LIN {X 0,Y 574.072,Z 399.932,A -85,B 0,C 180,E1 -2018.319,E2 -2018.319} C_VEL
LIN {X 0,Y 573.881,Z 501.404,A -85,B 0,C 180,E1 -2019.612,E2 -2019.612} C_VEL
LIN {X 0,Y 573.788,Z 514.414,A -85,B 0,C 180,E1 -2019.919,E2 -2019.919} C_VEL
LIN {X 0,Y 573.675,Z 527.236,A -85,B 0,C 180,E1 -2020.373,E2 -2020.373} C_VEL
LIN {X 0,Y 573.572,Z 539.532,A -85,B 0,C 180,E1 -2020.968,E2 -2020.968} C_VEL
LIN {X 0,Y 573.479,Z 550.065,A -85,B 0,C 180,E1 -2021.62,E2 -2021.62} C_VEL
LIN {X 0,Y 573.322,Z 560.171,A -85,B 0,C 180,E1 -2022.393,E2 -2022.393} C_VEL
LIN {X 0,Y 573.221,Z 570.379,A -85,B 0,C 180,E1 -2023.361,E2 -2023.361} C_VEL
LIN {X 0,Y 573.135,Z 578.736,A -85,B 0,C 180,E1 -2024.344,E2 -2024.344} C_VEL
LIN {X 0,Y 573.071,Z 585.667,A -85,B 0,C 180,E1 -2025.341,E2 -2025.341} C_VEL
LIN {X 0,Y 573.025,Z 591.385,A -85,B 0,C 180,E1 -2026.355,E2 -2026.355} C_VEL
LIN {X 0,Y 573.008,Z 596.786,A -85,B 0,C 180,E1 -2027.578,E2 -2027.578} C_VEL
LIN {X 0,Y 572.995,Z 599.936,A -85,B 0,C 180,E1 -2028.521,E2 -2028.521} C_VEL
LIN {X 0,Y 572.949,Z 602.391,A -85,B 0,C 180,E1 -2029.51,E2 -2029.51} C_VEL
LIN {X 0,Y 572.921,Z 604.15,A -85,B 0,C 180,E1 -2030.608,E2 -2030.608} C_VEL
LIN {X 0,Y 572.93,Z 604.936,A -85,B 0,C 180,E1 -2031.728,E2 -2031.728} C_VEL
LIN {X 0,Y 572.956,Z 604.58,A -85,B 0,C 180,E1 -2033.055,E2 -2033.055} C_VEL
LIN {X 0,Y 572.93,Z 603.35,A -85,B 0,C 180,E1 -2034.058,E2 -2034.058} C_VEL
LIN {X 0,Y 572.989,Z 600.789,A -85,B 0,C 180,E1 -2035.265,E2 -2035.265} C_VEL
LIN {X 0,Y 572.998,Z 596.77,A -85,B 0,C 180,E1 -2036.517,E2 -2036.517} C_VEL
LIN {X 0,Y 573.082,Z 591.054,A -85,B 0,C 180,E1 -2037.799,E2 -2037.799} C_VEL
LIN {X 0,Y 573.123,Z 584.06,A -85,B 0,C 180,E1 -2039,E2 -2039} C_VEL
LIN {X 0,Y 573.181,Z 576.654,A -85,B 0,C 180,E1 -2040.01,E2 -2040.01} C_VEL
LIN {X 0,Y 573.27,Z 567.371,A -85,B 0,C 180,E1 -2041.036,E2 -2041.036} C_VEL
LIN {X 0,Y 573.355,Z 557.054,A -85,B 0,C 180,E1 -2041.953,E2 -2041.953} C_VEL
LIN {X 0,Y 573.484,Z 545.995,A -85,B 0,C 180,E1 -2042.739,E2 -2042.739} C_VEL
LIN {X 0,Y 573.617,Z 535.091,A -85,B 0,C 180,E1 -2043.356,E2 -2043.356} C_VEL
LIN {X 0,Y 573.709,Z 523.101,A -85,B 0,C 180,E1 -2043.88,E2 -2043.88} C_VEL
LIN {X 0,Y 573.83,Z 510.167,A -85,B 0,C 180,E1 -2044.288,E2 -2044.288} C_VEL
LIN {X 0,Y 573.889,Z 497.236,A -85,B 0,C 180,E1 -2044.546,E2 -2044.546} C_VEL
LIN {X 0,Y 574.062,Z 398.701,A -85,B 0,C 180,E1 -2045.786,E2 -2045.786} C_VEL
LIN {X 0,Y 573.309,Z 394.131,A -85,B 0,C 180,E1 -2045.873,E2 -2045.873} C_VEL
LIN {X 0,Y 573.457,Z 376.545,A -85,B 0,C 180,E1 -2048.923,E2 -2048.923} C_VEL
LIN {X 0,Y 573.564,Z 362.34,A -85,B 0,C 180,E1 -2051.422,E2 -2051.422} C_VEL
LIN {X 0,Y 573.289,Z 360.075,A -85,B 0,C 180,E1 -2051.875,E2 -2051.875} C_VEL
LIN {X 0,Y 573.241,Z 360.081,A -85,B 0,C 180,E1 -2054.351,E2 -2054.351} C_VEL
LIN {X 0,Y 573.241,Z 360.084,A -85,B 0,C 180,E1 -2056.529,E2 -2056.529} C_VEL
LIN {X 0,Y 573.269,Z 360.077,A -85,B 0,C 180,E1 -2058.744,E2 -2058.744} C_VEL
LIN {X 0,Y 573.288,Z 360.068,A -85,B 0,C 180,E1 -2061.54,E2 -2061.54} C_VEL
LIN {X 0,Y 573.294,Z 360.076,A -85,B 0,C 180,E1 -2064.371,E2 -2064.371} C_VEL
LIN {X 0,Y 573.316,Z 360.067,A -85,B 0,C 180,E1 -2067.892,E2 -2067.892} C_VEL
LIN {X 0,Y 573.336,Z 360.066,A -85,B 0,C 180,E1 -2070.701,E2 -2070.701} C_VEL
LIN {X 0,Y 573.309,Z 360.068,A -85,B 0,C 180,E1 -2072.81,E2 -2072.81} C_VEL
LIN {X 0,Y 573.292,Z 360.069,A -85,B 0,C 180,E1 -2075.627,E2 -2075.627} C_VEL
LIN {X 0,Y 573.285,Z 360.074,A -85,B 0,C 180,E1 -2078.458,E2 -2078.458} C_VEL
LIN {X 0,Y 573.275,Z 360.07,A -85,B 0,C 180,E1 -2081.311,E2 -2081.311} C_VEL
LIN {X 0,Y 573.284,Z 360.073,A -85,B 0,C 180,E1 -2084.423,E2 -2084.423} C_VEL
LIN {X 0,Y 573.261,Z 360.071,A -85,B 0,C 180,E1 -2087.11,E2 -2087.11} C_VEL
LIN {X 0,Y 573.242,Z 360.082,A -85,B 0,C 180,E1 -2090.076,E2 -2090.076} C_VEL
LIN {X 0,Y 573.235,Z 360.078,A -85,B 0,C 180,E1 -2092.337,E2 -2092.337} C_VEL
LIN {X 0,Y 573.255,Z 360.075,A -85,B 0,C 180,E1 -2095.409,E2 -2095.409} C_VEL
LIN {X 0,Y 573.252,Z 360.079,A -85,B 0,C 180,E1 -2098.028,E2 -2098.028} C_VEL
LIN {X 0,Y 573.241,Z 360.074,A -85,B 0,C 180,E1 -2100.884,E2 -2100.884} C_VEL
LIN {X 0,Y 573.259,Z 360.079,A -85,B 0,C 180,E1 -2103.523,E2 -2103.523} C_VEL
LIN {X 0,Y 573.259,Z 360.075,A -85,B 0,C 180,E1 -2106.047,E2 -2106.047} C_VEL
LIN {X 0,Y 573.246,Z 360.073,A -85,B 0,C 180,E1 -2108.7,E2 -2108.7} C_VEL
LIN {X 0,Y 573.25,Z 360.082,A -85,B 0,C 180,E1 -2111.595,E2 -2111.595} C_VEL
LIN {X 0,Y 573.234,Z 360.076,A -85,B 0,C 180,E1 -2114.332,E2 -2114.332} C_VEL
LIN {X 0,Y 573.245,Z 360.083,A -85,B 0,C 180,E1 -2117.356,E2 -2117.356} C_VEL
LIN {X 0,Y 573.287,Z 360.256,A -85,B 0,C 180,E1 -2118.288,E2 -2118.288} C_VEL
LIN {X 0,Y 573.535,Z 365.736,A -85,B 0,C 180,E1 -2119.269,E2 -2119.269} C_VEL
LIN {X 0,Y 573.423,Z 380.934,A -85,B 0,C 180,E1 -2121.932,E2 -2121.932} C_VEL
LIN {X 0,Y 573.275,Z 394.135,A -85,B 0,C 180,E1 -2124.217,E2 -2124.217} C_VEL
LIN {X 0,Y 574.068,Z 400.409,A -85,B 0,C 180,E1 -2124.325,E2 -2124.325} C_VEL
LIN {X 0,Y 573.887,Z 500.332,A -85,B 0,C 180,E1 -2125.597,E2 -2125.597} C_VEL
LIN {X 0,Y 573.82,Z 512.126,A -85,B 0,C 180,E1 -2125.857,E2 -2125.857} C_VEL
LIN {X 0,Y 573.706,Z 525.236,A -85,B 0,C 180,E1 -2126.292,E2 -2126.292} C_VEL
LIN {X 0,Y 573.58,Z 537.36,A -85,B 0,C 180,E1 -2126.853,E2 -2126.853} C_VEL
LIN {X 0,Y 573.467,Z 548.11,A -85,B 0,C 180,E1 -2127.492,E2 -2127.492} C_VEL
LIN {X 0,Y 573.346,Z 558.978,A -85,B 0,C 180,E1 -2128.294,E2 -2128.294} C_VEL
LIN {X 0,Y 573.265,Z 569.447,A -85,B 0,C 180,E1 -2129.265,E2 -2129.265} C_VEL
LIN {X 0,Y 573.129,Z 577.631,A -85,B 0,C 180,E1 -2130.207,E2 -2130.207} C_VEL
LIN {X 0,Y 573.111,Z 584.91,A -85,B 0,C 180,E1 -2131.228,E2 -2131.228} C_VEL
LIN {X 0,Y 573.022,Z 591.708,A -85,B 0,C 180,E1 -2132.419,E2 -2132.419} C_VEL
LIN {X 0,Y 573.03,Z 596.673,A -85,B 0,C 180,E1 -2133.546,E2 -2133.546} C_VEL
LIN {X 0,Y 572.989,Z 600.113,A -85,B 0,C 180,E1 -2134.577,E2 -2134.577} C_VEL
LIN {X 0,Y 572.959,Z 602.073,A -85,B 0,C 180,E1 -2135.351,E2 -2135.351} C_VEL
LIN {X 0,Y 572.924,Z 603.479,A -85,B 0,C 180,E1 -2136.121,E2 -2136.121} C_VEL
LIN {X 0,Y 572.967,Z 604.451,A -85,B 0,C 180,E1 -2136.915,E2 -2136.915} C_VEL
LIN {X 0,Y 572.938,Z 604.921,A -85,B 0,C 180,E1 -2137.65,E2 -2137.65} C_VEL
LIN {X 0,Y 572.97,Z 604.761,A -85,B 0,C 180,E1 -2138.778,E2 -2138.778} C_VEL
LIN {X 0,Y 572.969,Z 603.567,A -85,B 0,C 180,E1 -2139.913,E2 -2139.913} C_VEL
LIN {X 0,Y 572.956,Z 601.885,A -85,B 0,C 180,E1 -2140.817,E2 -2140.817} C_VEL
LIN {X 0,Y 572.991,Z 599.33,A -85,B 0,C 180,E1 -2141.774,E2 -2141.774} C_VEL
LIN {X 0,Y 572.994,Z 595.309,A -85,B 0,C 180,E1 -2142.88,E2 -2142.88} C_VEL
LIN {X 0,Y 573.044,Z 590.075,A -85,B 0,C 180,E1 -2143.981,E2 -2143.981} C_VEL
LIN {X 0,Y 573.091,Z 583.522,A -85,B 0,C 180,E1 -2145.076,E2 -2145.076} C_VEL
LIN {X 0,Y 573.174,Z 575.367,A -85,B 0,C 180,E1 -2146.166,E2 -2146.166} C_VEL
LIN {X 0,Y 573.277,Z 567.009,A -85,B 0,C 180,E1 -2147.071,E2 -2147.071} C_VEL
LIN {X 0,Y 573.342,Z 557.888,A -85,B 0,C 180,E1 -2147.882,E2 -2147.882} C_VEL
LIN {X 0,Y 573.449,Z 548.891,A -85,B 0,C 180,E1 -2148.546,E2 -2148.546} C_VEL
LIN {X 0,Y 573.551,Z 538.875,A -85,B 0,C 180,E1 -2149.154,E2 -2149.154} C_VEL
LIN {X 0,Y 573.661,Z 528.069,A -85,B 0,C 180,E1 -2149.678,E2 -2149.678} C_VEL
LIN {X 0,Y 573.77,Z 515.206,A -85,B 0,C 180,E1 -2150.148,E2 -2150.148} C_VEL
LIN {X 0,Y 573.895,Z 502.194,A -85,B 0,C 180,E1 -2150.462,E2 -2150.462} C_VEL
LIN {X 0,Y 573.934,Z 468.796,A -85,B 0,C 180,E1 -2150.907,E2 -2150.907} C_VEL
LIN {X 0,Y 574.041,Z 398.761,A -85,B 0,C 180,E1 -2151.786,E2 -2151.786} C_VEL
LIN {X 0,Y 573.334,Z 394.179,A -85,B 0,C 180,E1 -2151.864,E2 -2151.864} C_VEL
LIN {X 0,Y 573.428,Z 376.67,A -85,B 0,C 180,E1 -2154.902,E2 -2154.902} C_VEL
LIN {X 0,Y 573.566,Z 363.645,A -85,B 0,C 180,E1 -2157.191,E2 -2157.191} C_VEL
LIN {X 0,Y 573.275,Z 360.076,A -85,B 0,C 180,E1 -2157.848,E2 -2157.848} C_VEL
LIN {X 0,Y 573.312,Z 360.069,A -85,B 0,C 180,E1 -2160,E2 -2160} C_VEL
LIN {X 0,Y 573.306,Z 360.073,A -85,B 0,C 180,E1 -2162.811,E2 -2162.811} C_VEL
LIN {X 0,Y 573.285,Z 360.07,A -85,B 0,C 180,E1 -2165.628,E2 -2165.628} C_VEL
LIN {X 0,Y 573.298,Z 360.076,A -85,B 0,C 180,E1 -2168.459,E2 -2168.459} C_VEL
LIN {X 0,Y 573.289,Z 360.069,A -85,B 0,C 180,E1 -2171.312,E2 -2171.312} C_VEL
LIN {X 0,Y 573.271,Z 360.077,A -85,B 0,C 180,E1 -2174.425,E2 -2174.425} C_VEL
LIN {X 0,Y 573.252,Z 360.073,A -85,B 0,C 180,E1 -2177.112,E2 -2177.112} C_VEL
LIN {X 0,Y 573.25,Z 360.082,A -85,B 0,C 180,E1 -2180.077,E2 -2180.077} C_VEL
LIN {X 0,Y 573.262,Z 360.072,A -85,B 0,C 180,E1 -2183.154,E2 -2183.154} C_VEL
LIN {X 0,Y 573.284,Z 360.073,A -85,B 0,C 180,E1 -2186.189,E2 -2186.189} C_VEL
LIN {X 0,Y 573.235,Z 360.076,A -85,B 0,C 180,E1 -2188.565,E2 -2188.565} C_VEL
LIN {X 0,Y 573.234,Z 360.077,A -85,B 0,C 180,E1 -2190.993,E2 -2190.993} C_VEL
LIN {X 0,Y 573.28,Z 360.079,A -85,B 0,C 180,E1 -2193.529,E2 -2193.529} C_VEL
LIN {X 0,Y 573.253,Z 360.075,A -85,B 0,C 180,E1 -2196.049,E2 -2196.049} C_VEL
LIN {X 0,Y 573.242,Z 360.075,A -85,B 0,C 180,E1 -2198.702,E2 -2198.702} C_VEL
LIN {X 0,Y 573.247,Z 360.079,A -85,B 0,C 180,E1 -2201.597,E2 -2201.597} C_VEL
LIN {X 0,Y 573.233,Z 360.075,A -85,B 0,C 180,E1 -2204.334,E2 -2204.334} C_VEL
LIN {X 0,Y 573.234,Z 360.082,A -85,B 0,C 180,E1 -2207.359,E2 -2207.359} C_VEL
LIN {X 0,Y 573.244,Z 360.075,A -85,B 0,C 180,E1 -2210.394,E2 -2210.394} C_VEL
LIN {X 0,Y 573.253,Z 360.081,A -85,B 0,C 180,E1 -2213.079,E2 -2213.079} C_VEL
LIN {X 0,Y 573.272,Z 360.071,A -85,B 0,C 180,E1 -2215.673,E2 -2215.673} C_VEL
LIN {X 0,Y 573.247,Z 360.075,A -85,B 0,C 180,E1 -2218.186,E2 -2218.186} C_VEL
LIN {X 0,Y 573.268,Z 360.079,A -85,B 0,C 180,E1 -2220.636,E2 -2220.636} C_VEL
LIN {X 0,Y 573.269,Z 360.072,A -85,B 0,C 180,E1 -2223.502,E2 -2223.502} C_VEL
LIN {X 0,Y 573.232,Z 360.081,A -85,B 0,C 180,E1 -2226.136,E2 -2226.136} C_VEL
LIN {X 0,Y 573.254,Z 360.175,A -85,B 0,C 180,E1 -2226.937,E2 -2226.937} C_VEL
LIN {X 0,Y 574.015,Z 365.028,A -85,B 0,C 180,E1 -2227.695,E2 -2227.695} C_VEL
LIN {X 0,Y 573.747,Z 385.178,A -85,B 0,C 180,E1 -2230.688,E2 -2230.688} C_VEL
LIN {X 0,Y 573.562,Z 404.099,A -85,B 0,C 180,E1 -2233.454,E2 -2233.454} C_VEL
LIN {X 0,Y 573.381,Z 422.8,A -85,B 0,C 180,E1 -2236.15,E2 -2236.15} C_VEL
LIN {X 0,Y 574.12,Z 428.592,A -85,B 0,C 180,E1 -2236.259,E2 -2236.259} C_VEL
LIN {X 0,Y 573.908,Z 530.999,A -85,B 0,C 180,E1 -2237.559,E2 -2237.559} C_VEL
LIN {X 0,Y 573.777,Z 544.254,A -85,B 0,C 180,E1 -2237.87,E2 -2237.87} C_VEL
LIN {X 0,Y 573.703,Z 556.4,A -85,B 0,C 180,E1 -2238.295,E2 -2238.295} C_VEL
LIN {X 0,Y 573.593,Z 568.646,A -85,B 0,C 180,E1 -2238.874,E2 -2238.874} C_VEL
LIN {X 0,Y 573.434,Z 580.216,A -85,B 0,C 180,E1 -2239.586,E2 -2239.586} C_VEL
LIN {X 0,Y 573.327,Z 590.612,A -85,B 0,C 180,E1 -2240.386,E2 -2240.386} C_VEL
LIN {X 0,Y 573.24,Z 599.123,A -85,B 0,C 180,E1 -2241.186,E2 -2241.186} C_VEL
LIN {X 0,Y 573.16,Z 606.969,A -85,B 0,C 180,E1 -2242.072,E2 -2242.072} C_VEL
LIN {X 0,Y 573.073,Z 614.586,A -85,B 0,C 180,E1 -2243.127,E2 -2243.127} C_VEL
LIN {X 0,Y 573.07,Z 621.685,A -85,B 0,C 180,E1 -2244.371,E2 -2244.371} C_VEL
LIN {X 0,Y 573.028,Z 626.376,A -85,B 0,C 180,E1 -2245.428,E2 -2245.428} C_VEL
LIN {X 0,Y 573.022,Z 629.96,A -85,B 0,C 180,E1 -2246.485,E2 -2246.485} C_VEL
LIN {X 0,Y 572.959,Z 631.81,A -85,B 0,C 180,E1 -2247.189,E2 -2247.189} C_VEL
LIN {X 0,Y 572.938,Z 633.2,A -85,B 0,C 180,E1 -2247.892,E2 -2247.892} C_VEL
LIN {X 0,Y 572.941,Z 634.786,A -85,B 0,C 180,E1 -2249.298,E2 -2249.298} C_VEL
LIN {X 0,Y 572.938,Z 635,A -85,B 0,C 180,E1 -2250.001,E2 -2250.001} C_VEL
LIN {X 0,Y 572.946,Z 634.185,A -85,B 0,C 180,E1 -2251.407,E2 -2251.407} C_VEL
LIN {X 0,Y 572.938,Z 633.198,A -85,B 0,C 180,E1 -2252.11,E2 -2252.11} C_VEL
LIN {X 0,Y 572.959,Z 631.808,A -85,B 0,C 180,E1 -2252.813,E2 -2252.813} C_VEL
LIN {X 0,Y 573.014,Z 628.893,A -85,B 0,C 180,E1 -2253.869,E2 -2253.869} C_VEL
LIN {X 0,Y 572.963,Z 624.945,A -85,B 0,C 180,E1 -2254.926,E2 -2254.926} C_VEL
LIN {X 0,Y 573.064,Z 618.872,A -85,B 0,C 180,E1 -2256.161,E2 -2256.161} C_VEL
LIN {X 0,Y 573.12,Z 612.232,A -85,B 0,C 180,E1 -2257.222,E2 -2257.222} C_VEL
LIN {X 0,Y 573.199,Z 603.983,A -85,B 0,C 180,E1 -2258.284,E2 -2258.284} C_VEL
LIN {X 0,Y 573.287,Z 595.529,A -85,B 0,C 180,E1 -2259.171,E2 -2259.171} C_VEL
LIN {X 0,Y 573.421,Z 585.087,A -85,B 0,C 180,E1 -2260.059,E2 -2260.059} C_VEL
LIN {X 0,Y 573.528,Z 573.342,A -85,B 0,C 180,E1 -2260.859,E2 -2260.859} C_VEL
LIN {X 0,Y 573.655,Z 562.264,A -85,B 0,C 180,E1 -2261.448,E2 -2261.448} C_VEL
LIN {X 0,Y 573.759,Z 549.148,A -85,B 0,C 180,E1 -2261.975,E2 -2261.975} C_VEL
LIN {X 0,Y 573.866,Z 536.485,A -85,B 0,C 180,E1 -2262.331,E2 -2262.331} C_VEL
LIN {X 0,Y 573.928,Z 523.244,A -85,B 0,C 180,E1 -2262.555,E2 -2262.555} C_VEL
LIN {X 0,Y 573.944,Z 426.655,A -85,B 0,C 180,E1 -2263.77,E2 -2263.77} C_VEL
LIN {X 0,Y 573.379,Z 422.787,A -85,B 0,C 180,E1 -2263.852,E2 -2263.852} C_VEL
LIN {X 0,Y 573.547,Z 402.884,A -85,B 0,C 180,E1 -2266.724,E2 -2266.724} C_VEL
LIN {X 0,Y 573.735,Z 384.58,A -85,B 0,C 180,E1 -2269.401,E2 -2269.401} C_VEL
LIN {X 0,Y 574.002,Z 365.015,A -85,B 0,C 180,E1 -2272.307,E2 -2272.307} C_VEL
LIN {X 0,Y 573.24,Z 360.085,A -85,B 0,C 180,E1 -2273.1,E2 -2273.1} C_VEL
LIN {X 0,Y 573.261,Z 360.081,A -85,B 0,C 180,E1 -2275.411,E2 -2275.411} C_VEL
LIN {X 0,Y 573.256,Z 360.075,A -85,B 0,C 180,E1 -2278.029,E2 -2278.029} C_VEL
LIN {X 0,Y 573.244,Z 360.079,A -85,B 0,C 180,E1 -2280.884,E2 -2280.884} C_VEL
LIN {X 0,Y 573.268,Z 360.076,A -85,B 0,C 180,E1 -2283.524,E2 -2283.524} C_VEL
LIN {X 0,Y 573.221,Z 360.077,A -85,B 0,C 180,E1 -2286.052,E2 -2286.052} C_VEL
LIN {X 0,Y 573.255,Z 360.077,A -85,B 0,C 180,E1 -2288.701,E2 -2288.701} C_VEL
LIN {X 0,Y 573.234,Z 360.078,A -85,B 0,C 180,E1 -2291.593,E2 -2291.593} C_VEL
LIN {X 0,Y 573.241,Z 360.076,A -85,B 0,C 180,E1 -2294.334,E2 -2294.334} C_VEL
LIN {X 0,Y 573.246,Z 360.077,A -85,B 0,C 180,E1 -2297.359,E2 -2297.359} C_VEL
LIN {X 0,Y 573.243,Z 360.076,A -85,B 0,C 180,E1 -2300.392,E2 -2300.392} C_VEL
LIN {X 0,Y 573.257,Z 360.078,A -85,B 0,C 180,E1 -2303.078,E2 -2303.078} C_VEL
LIN {X 0,Y 573.271,Z 360.07,A -85,B 0,C 180,E1 -2305.671,E2 -2305.671} C_VEL
LIN {X 0,Y 573.245,Z 360.076,A -85,B 0,C 180,E1 -2308.185,E2 -2308.185} C_VEL
LIN {X 0,Y 573.268,Z 360.079,A -85,B 0,C 180,E1 -2310.634,E2 -2310.634} C_VEL
LIN {X 0,Y 573.24,Z 360.073,A -85,B 0,C 180,E1 -2313.508,E2 -2313.508} C_VEL
LIN {X 0,Y 573.235,Z 360.078,A -85,B 0,C 180,E1 -2316.135,E2 -2316.135} C_VEL
LIN {X 0,Y 573.255,Z 360.074,A -85,B 0,C 180,E1 -2319.174,E2 -2319.174} C_VEL
LIN {X 0,Y 573.222,Z 360.075,A -85,B 0,C 180,E1 -2321.411,E2 -2321.411} C_VEL
LIN {X 0,Y 573.254,Z 360.073,A -85,B 0,C 180,E1 -2323.622,E2 -2323.622} C_VEL
LIN {X 0,Y 573.277,Z 360.07,A -85,B 0,C 180,E1 -2325.807,E2 -2325.807} C_VEL
LIN {X 0,Y 573.269,Z 360.073,A -85,B 0,C 180,E1 -2328.745,E2 -2328.745} C_VEL
LIN {X 0,Y 573.288,Z 360.069,A -85,B 0,C 180,E1 -2331.541,E2 -2331.541} C_VEL
LIN {X 0,Y 573.295,Z 360.074,A -85,B 0,C 180,E1 -2334.372,E2 -2334.372} C_VEL
LIN {X 0,Y 573.316,Z 360.07,A -85,B 0,C 180,E1 -2337.892,E2 -2337.892} C_VEL
LIN {X 0,Y 573.335,Z 360.063,A -85,B 0,C 180,E1 -2340.702,E2 -2340.702} C_VEL
LIN {X 0,Y 573.311,Z 360.066,A -85,B 0,C 180,E1 -2342.811,E2 -2342.811} C_VEL
LIN {X 0,Y 573.296,Z 360.072,A -85,B 0,C 180,E1 -2345.628,E2 -2345.628} C_VEL
LIN {X 0,Y 573.289,Z 360.07,A -85,B 0,C 180,E1 -2348.46,E2 -2348.46} C_VEL
LIN {X 0,Y 573.278,Z 360.072,A -85,B 0,C 180,E1 -2351.312,E2 -2351.312} C_VEL
LIN {X 0,Y 573.287,Z 360.07,A -85,B 0,C 180,E1 -2354.424,E2 -2354.424} C_VEL
LIN {X 0,Y 573.264,Z 360.073,A -85,B 0,C 180,E1 -2357.112,E2 -2357.112} C_VEL
LIN {X 0,Y 573.257,Z 360.076,A -85,B 0,C 180,E1 -2360.077,E2 -2360.077} C_VEL
LIN {X 0,Y 573.241,Z 360.077,A -85,B 0,C 180,E1 -2363.099,E2 -2363.099} C_VEL
LIN {X 0,Y 573.255,Z 360.073,A -85,B 0,C 180,E1 -2364.387,E2 -2364.387} C_VEL
LIN {X 0,Y 572.63,Z 360.154,A -85,B 0,C 180,E1 -2364.974,E2 -2364.974} C_VEL
LIN {X 0,Y 569.791,Z 360.512,A -85,B 0,C 180,E1 -2365.925,E2 -2365.925} C_VEL
LIN {X 0,Y 567.357,Z 360.818,A -85,B 0,C 180,E1 -2366.691,E2 -2366.691} C_VEL
LIN {X 0,Y 566.296,Z 360.948,A -85,B 0,C 180,E1 -2367.282,E2 -2367.282} C_VEL
LIN {X 0,Y 566.203,Z 360.957,A -85,B 0,C 180,E1 -2367.482,E2 -2367.482} C_VEL
LIN {X 0,Y 566.207,Z 360.958,A -85,B 0,C 180,E1 -2369.769,E2 -2369.769} C_VEL
LIN {X 0,Y 566.23,Z 361.071,A -85,B 0,C 180,E1 -2372.178,E2 -2372.178} C_VEL
LIN {X 0,Y 566.543,Z 366.033,A -85,B 0,C 180,E1 -2373.081,E2 -2373.081} C_VEL
LIN {X 0,Y 566.377,Z 382.226,A -85,B 0,C 180,E1 -2375.954,E2 -2375.954} C_VEL
LIN {X 0,Y 566.257,Z 394.162,A -85,B 0,C 180,E1 -2378.047,E2 -2378.047} C_VEL
LIN {X 0,Y 567.172,Z 400.604,A -85,B 0,C 180,E1 -2378.158,E2 -2378.158} C_VEL
LIN {X 0,Y 566.943,Z 501.598,A -85,B 0,C 180,E1 -2379.461,E2 -2379.461} C_VEL
LIN {X 0,Y 566.835,Z 514.735,A -85,B 0,C 180,E1 -2379.778,E2 -2379.778} C_VEL
LIN {X 0,Y 566.716,Z 526.907,A -85,B 0,C 180,E1 -2380.214,E2 -2380.214} C_VEL
LIN {X 0,Y 566.595,Z 539.544,A -85,B 0,C 180,E1 -2380.83,E2 -2380.83} C_VEL
LIN {X 0,Y 566.465,Z 551.449,A -85,B 0,C 180,E1 -2381.588,E2 -2381.588} C_VEL
LIN {X 0,Y 566.258,Z 562.13,A -85,B 0,C 180,E1 -2382.444,E2 -2382.444} C_VEL
LIN {X 0,Y 566.182,Z 570.576,A -85,B 0,C 180,E1 -2383.273,E2 -2383.273} C_VEL
LIN {X 0,Y 566.078,Z 578.913,A -85,B 0,C 180,E1 -2384.27,E2 -2384.27} C_VEL
LIN {X 0,Y 566.011,Z 585.787,A -85,B 0,C 180,E1 -2385.276,E2 -2385.276} C_VEL
LIN {X 0,Y 565.945,Z 592.441,A -85,B 0,C 180,E1 -2386.498,E2 -2386.498} C_VEL
LIN {X 0,Y 565.914,Z 596.69,A -85,B 0,C 180,E1 -2387.497,E2 -2387.497} C_VEL
LIN {X 0,Y 565.923,Z 599.027,A -85,B 0,C 180,E1 -2388.17,E2 -2388.17} C_VEL
LIN {X 0,Y 565.846,Z 601.944,A -85,B 0,C 180,E1 -2389.257,E2 -2389.257} C_VEL
LIN {X 0,Y 565.852,Z 603.889,A -85,B 0,C 180,E1 -2390.359,E2 -2390.359} C_VEL
LIN {X 0,Y 565.835,Z 604.911,A -85,B 0,C 180,E1 -2391.608,E2 -2391.608} C_VEL
LIN {X 0,Y 565.816,Z 604.853,A -85,B 0,C 180,E1 -2392.65,E2 -2392.65} C_VEL
LIN {X 0,Y 565.826,Z 603.728,A -85,B 0,C 180,E1 -2393.838,E2 -2393.838} C_VEL
LIN {X 0,Y 565.879,Z 601.155,A -85,B 0,C 180,E1 -2395.158,E2 -2395.158} C_VEL
LIN {X 0,Y 565.925,Z 597.713,A -85,B 0,C 180,E1 -2396.31,E2 -2396.31} C_VEL
LIN {X 0,Y 565.951,Z 592.347,A -85,B 0,C 180,E1 -2397.611,E2 -2397.611} C_VEL
LIN {X 0,Y 566.001,Z 585.959,A -85,B 0,C 180,E1 -2398.785,E2 -2398.785} C_VEL
LIN {X 0,Y 566.104,Z 578.954,A -85,B 0,C 180,E1 -2399.814,E2 -2399.814} C_VEL
LIN {X 0,Y 566.197,Z 570.325,A -85,B 0,C 180,E1 -2400.843,E2 -2400.843} C_VEL
LIN {X 0,Y 566.309,Z 560.612,A -85,B 0,C 180,E1 -2401.779,E2 -2401.779} C_VEL
LIN {X 0,Y 566.444,Z 550.474,A -85,B 0,C 180,E1 -2402.572,E2 -2402.572} C_VEL
LIN {X 0,Y 566.614,Z 539.526,A -85,B 0,C 180,E1 -2403.26,E2 -2403.26} C_VEL
LIN {X 0,Y 566.724,Z 527.948,A -85,B 0,C 180,E1 -2403.831,E2 -2403.831} C_VEL
LIN {X 0,Y 566.842,Z 515.148,A -85,B 0,C 180,E1 -2404.3,E2 -2404.3} C_VEL
LIN {X 0,Y 566.944,Z 502.434,A -85,B 0,C 180,E1 -2404.613,E2 -2404.613} C_VEL
LIN {X 0,Y 567.034,Z 471.171,A -85,B 0,C 180,E1 -2405.036,E2 -2405.036} C_VEL
LIN {X 0,Y 567.071,Z 399.012,A -85,B 0,C 180,E1 -2405.955,E2 -2405.955} C_VEL
LIN {X 0,Y 566.29,Z 394.166,A -85,B 0,C 180,E1 -2406.042,E2 -2406.042} C_VEL
LIN {X 0,Y 566.425,Z 376.763,A -85,B 0,C 180,E1 -2409.1,E2 -2409.1} C_VEL
LIN {X 0,Y 566.576,Z 364.003,A -85,B 0,C 180,E1 -2411.372,E2 -2411.372} C_VEL
LIN {X 0,Y 566.26,Z 360.951,A -85,B 0,C 180,E1 -2411.97,E2 -2411.97} C_VEL
LIN {X 0,Y 566.205,Z 360.957,A -85,B 0,C 180,E1 -2414.89,E2 -2414.89} C_VEL
LIN {X 0,Y 566.249,Z 360.946,A -85,B 0,C 180,E1 -2417.818,E2 -2417.818} C_VEL
LIN {X 0,Y 566.212,Z 360.956,A -85,B 0,C 180,E1 -2420.713,E2 -2420.713} C_VEL
LIN {X 0,Y 566.23,Z 360.948,A -85,B 0,C 180,E1 -2423.197,E2 -2423.197} C_VEL
LIN {X 0,Y 566.189,Z 360.953,A -85,B 0,C 180,E1 -2425.728,E2 -2425.728} C_VEL
LIN {X 0,Y 566.287,Z 360.943,A -85,B 0,C 180,E1 -2427.865,E2 -2427.865} C_VEL
LIN {X 0,Y 566.307,Z 360.942,A -85,B 0,C 180,E1 -2430.71,E2 -2430.71} C_VEL
LIN {X 0,Y 566.275,Z 360.944,A -85,B 0,C 180,E1 -2432.845,E2 -2432.845} C_VEL
LIN {X 0,Y 566.261,Z 360.946,A -85,B 0,C 180,E1 -2435.697,E2 -2435.697} C_VEL
LIN {X 0,Y 566.229,Z 360.951,A -85,B 0,C 180,E1 -2438.565,E2 -2438.565} C_VEL
LIN {X 0,Y 566.245,Z 360.947,A -85,B 0,C 180,E1 -2441.453,E2 -2441.453} C_VEL
LIN {X 0,Y 566.237,Z 360.95,A -85,B 0,C 180,E1 -2444.506,E2 -2444.506} C_VEL
LIN {X 0,Y 566.204,Z 360.952,A -85,B 0,C 180,E1 -2447.33,E2 -2447.33} C_VEL
LIN {X 0,Y 566.208,Z 360.954,A -85,B 0,C 180,E1 -2450.336,E2 -2450.336} C_VEL
LIN {X 0,Y 566.173,Z 360.956,A -85,B 0,C 180,E1 -2453.281,E2 -2453.281} C_VEL
LIN {X 0,Y 566.214,Z 360.958,A -85,B 0,C 180,E1 -2455.748,E2 -2455.748} C_VEL
LIN {X 0,Y 566.201,Z 360.954,A -85,B 0,C 180,E1 -2458.201,E2 -2458.201} C_VEL
LIN {X 0,Y 566.192,Z 360.952,A -85,B 0,C 180,E1 -2460.591,E2 -2460.591} C_VEL
LIN {X 0,Y 566.226,Z 360.949,A -85,B 0,C 180,E1 -2463.1,E2 -2463.1} C_VEL
LIN {X 0,Y 566.211,Z 360.959,A -85,B 0,C 180,E1 -2465.687,E2 -2465.687} C_VEL
LIN {X 0,Y 566.212,Z 360.949,A -85,B 0,C 180,E1 -2468.558,E2 -2468.558} C_VEL
LIN {X 0,Y 566.208,Z 360.954,A -85,B 0,C 180,E1 -2471.135,E2 -2471.135} C_VEL
LIN {X 0,Y 566.195,Z 360.955,A -85,B 0,C 180,E1 -2474.034,E2 -2474.034} C_VEL
LIN {X 0,Y 566.204,Z 360.956,A -85,B 0,C 180,E1 -2477.081,E2 -2477.081} C_VEL
LIN {X 0,Y 566.277,Z 361.149,A -85,B 0,C 180,E1 -2478.194,E2 -2478.194} C_VEL
LIN {X 0,Y 566.541,Z 366.546,A -85,B 0,C 180,E1 -2479.173,E2 -2479.173} C_VEL
LIN {X 0,Y 566.374,Z 383.071,A -85,B 0,C 180,E1 -2482.103,E2 -2482.103} C_VEL
LIN {X 0,Y 566.263,Z 394.133,A -85,B 0,C 180,E1 -2484.042,E2 -2484.042} C_VEL
LIN {X 0,Y 567.178,Z 399.933,A -85,B 0,C 180,E1 -2484.149,E2 -2484.149} C_VEL
LIN {X 0,Y 566.957,Z 500.764,A -85,B 0,C 180,E1 -2485.45,E2 -2485.45} C_VEL
LIN {X 0,Y 566.857,Z 513.412,A -85,B 0,C 180,E1 -2485.739,E2 -2485.739} C_VEL
LIN {X 0,Y 566.749,Z 526.141,A -85,B 0,C 180,E1 -2486.182,E2 -2486.182} C_VEL
LIN {X 0,Y 566.609,Z 537.294,A -85,B 0,C 180,E1 -2486.711,E2 -2486.711} C_VEL
LIN {X 0,Y 566.469,Z 548.004,A -85,B 0,C 180,E1 -2487.354,E2 -2487.354} C_VEL
LIN {X 0,Y 566.325,Z 557.62,A -85,B 0,C 180,E1 -2488.064,E2 -2488.064} C_VEL
LIN {X 0,Y 566.22,Z 567.122,A -85,B 0,C 180,E1 -2488.916,E2 -2488.916} C_VEL
LIN {X 0,Y 566.096,Z 576.945,A -85,B 0,C 180,E1 -2490.02,E2 -2490.02} C_VEL
LIN {X 0,Y 566.037,Z 584.23,A -85,B 0,C 180,E1 -2491.038,E2 -2491.038} C_VEL
LIN {X 0,Y 565.942,Z 590.121,A -85,B 0,C 180,E1 -2492.044,E2 -2492.044} C_VEL
LIN {X 0,Y 565.928,Z 594.856,A -85,B 0,C 180,E1 -2493.046,E2 -2493.046} C_VEL
LIN {X 0,Y 565.918,Z 599.224,A -85,B 0,C 180,E1 -2494.236,E2 -2494.236} C_VEL
LIN {X 0,Y 565.861,Z 601.399,A -85,B 0,C 180,E1 -2495.045,E2 -2495.045} C_VEL
LIN {X 0,Y 565.827,Z 602.987,A -85,B 0,C 180,E1 -2495.802,E2 -2495.802} C_VEL
LIN {X 0,Y 565.845,Z 604.354,A -85,B 0,C 180,E1 -2496.792,E2 -2496.792} C_VEL
LIN {X 0,Y 565.83,Z 604.952,A -85,B 0,C 180,E1 -2498.122,E2 -2498.122} C_VEL
LIN {X 0,Y 565.884,Z 604.688,A -85,B 0,C 180,E1 -2498.889,E2 -2498.889} C_VEL
LIN {X 0,Y 565.855,Z 603.994,A -85,B 0,C 180,E1 -2499.649,E2 -2499.649} C_VEL
LIN {X 0,Y 565.863,Z 602.194,A -85,B 0,C 180,E1 -2500.716,E2 -2500.716} C_VEL
LIN {X 0,Y 565.908,Z 599.027,A -85,B 0,C 180,E1 -2501.912,E2 -2501.912} C_VEL
LIN {X 0,Y 565.922,Z 595.122,A -85,B 0,C 180,E1 -2502.982,E2 -2502.982} C_VEL
LIN {X 0,Y 565.95,Z 589.593,A -85,B 0,C 180,E1 -2504.145,E2 -2504.145} C_VEL
LIN {X 0,Y 566.043,Z 582.7,A -85,B 0,C 180,E1 -2505.291,E2 -2505.291} C_VEL
LIN {X 0,Y 566.118,Z 574.637,A -85,B 0,C 180,E1 -2506.357,E2 -2506.357} C_VEL
LIN {X 0,Y 566.239,Z 566.073,A -85,B 0,C 180,E1 -2507.273,E2 -2507.273} C_VEL
LIN {X 0,Y 566.342,Z 556.77,A -85,B 0,C 180,E1 -2508.094,E2 -2508.094} C_VEL
LIN {X 0,Y 566.445,Z 548.159,A -85,B 0,C 180,E1 -2508.726,E2 -2508.726} C_VEL
LIN {X 0,Y 566.643,Z 537.477,A -85,B 0,C 180,E1 -2509.368,E2 -2509.368} C_VEL
LIN {X 0,Y 566.774,Z 524.897,A -85,B 0,C 180,E1 -2509.958,E2 -2509.958} C_VEL
LIN {X 0,Y 566.842,Z 512.035,A -85,B 0,C 180,E1 -2510.387,E2 -2510.387} C_VEL
LIN {X 0,Y 566.96,Z 500.947,A -85,B 0,C 180,E1 -2510.636,E2 -2510.636} C_VEL
LIN {X 0,Y 567.087,Z 399.252,A -85,B 0,C 180,E1 -2511.952,E2 -2511.952} C_VEL
LIN {X 0,Y 566.276,Z 394.042,A -85,B 0,C 180,E1 -2512.064,E2 -2512.064} C_VEL
LIN {X 0,Y 566.403,Z 377.236,A -85,B 0,C 180,E1 -2515.017,E2 -2515.017} C_VEL
LIN {X 0,Y 566.571,Z 365.207,A -85,B 0,C 180,E1 -2517.156,E2 -2517.156} C_VEL
LIN {X 0,Y 566.266,Z 360.949,A -85,B 0,C 180,E1 -2517.955,E2 -2517.955} C_VEL
LIN {X 0,Y 566.3,Z 360.948,A -85,B 0,C 180,E1 -2520.711,E2 -2520.711} C_VEL
LIN {X 0,Y 566.271,Z 360.949,A -85,B 0,C 180,E1 -2522.846,E2 -2522.846} C_VEL
LIN {X 0,Y 566.253,Z 360.947,A -85,B 0,C 180,E1 -2525.698,E2 -2525.698} C_VEL
LIN {X 0,Y 566.239,Z 360.953,A -85,B 0,C 180,E1 -2528.566,E2 -2528.566} C_VEL
LIN {X 0,Y 566.241,Z 360.947,A -85,B 0,C 180,E1 -2531.454,E2 -2531.454} C_VEL
LIN {X 0,Y 566.224,Z 360.953,A -85,B 0,C 180,E1 -2534.507,E2 -2534.507} C_VEL
LIN {X 0,Y 566.197,Z 360.953,A -85,B 0,C 180,E1 -2537.332,E2 -2537.332} C_VEL
LIN {X 0,Y 566.212,Z 360.954,A -85,B 0,C 180,E1 -2540.337,E2 -2540.337} C_VEL
LIN {X 0,Y 566.225,Z 360.951,A -85,B 0,C 180,E1 -2543.402,E2 -2543.402} C_VEL
LIN {X 0,Y 566.22,Z 360.958,A -85,B 0,C 180,E1 -2545.749,E2 -2545.749} C_VEL
LIN {X 0,Y 566.199,Z 360.955,A -85,B 0,C 180,E1 -2548.204,E2 -2548.204} C_VEL
LIN {X 0,Y 566.187,Z 360.953,A -85,B 0,C 180,E1 -2550.593,E2 -2550.593} C_VEL
LIN {X 0,Y 566.221,Z 360.952,A -85,B 0,C 180,E1 -2553.102,E2 -2553.102} C_VEL
LIN {X 0,Y 566.204,Z 360.958,A -85,B 0,C 180,E1 -2555.689,E2 -2555.689} C_VEL
LIN {X 0,Y 566.208,Z 360.951,A -85,B 0,C 180,E1 -2558.56,E2 -2558.56} C_VEL
LIN {X 0,Y 566.205,Z 360.957,A -85,B 0,C 180,E1 -2561.137,E2 -2561.137} C_VEL
LIN {X 0,Y 566.194,Z 360.953,A -85,B 0,C 180,E1 -2564.036,E2 -2564.036} C_VEL
LIN {X 0,Y 566.195,Z 360.96,A -85,B 0,C 180,E1 -2567.084,E2 -2567.084} C_VEL
LIN {X 0,Y 566.222,Z 360.95,A -85,B 0,C 180,E1 -2569.804,E2 -2569.804} C_VEL
LIN {X 0,Y 566.195,Z 360.956,A -85,B 0,C 180,E1 -2572.6,E2 -2572.6} C_VEL
LIN {X 0,Y 566.219,Z 360.955,A -85,B 0,C 180,E1 -2575.184,E2 -2575.184} C_VEL
LIN {X 0,Y 566.231,Z 360.948,A -85,B 0,C 180,E1 -2577.745,E2 -2577.745} C_VEL
LIN {X 0,Y 566.226,Z 360.952,A -85,B 0,C 180,E1 -2580.324,E2 -2580.324} C_VEL
LIN {X 0,Y 566.233,Z 360.95,A -85,B 0,C 180,E1 -2583.336,E2 -2583.336} C_VEL
LIN {X 0,Y 566.198,Z 360.955,A -85,B 0,C 180,E1 -2585.821,E2 -2585.821} C_VEL
LIN {X 0,Y 566.208,Z 361.122,A -85,B 0,C 180,E1 -2586.798,E2 -2586.798} C_VEL
LIN {X 0,Y 567.07,Z 366.19,A -85,B 0,C 180,E1 -2587.599,E2 -2587.599} C_VEL
LIN {X 0,Y 566.788,Z 386.047,A -85,B 0,C 180,E1 -2590.571,E2 -2590.571} C_VEL
LIN {X 0,Y 566.58,Z 404.253,A -85,B 0,C 180,E1 -2593.266,E2 -2593.266} C_VEL
LIN {X 0,Y 566.386,Z 422.8,A -85,B 0,C 180,E1 -2595.976,E2 -2595.976} C_VEL
LIN {X 0,Y 567.214,Z 429.374,A -85,B 0,C 180,E1 -2596.098,E2 -2596.098} C_VEL
LIN {X 0,Y 566.988,Z 530.999,A -85,B 0,C 180,E1 -2597.405,E2 -2597.405} C_VEL
LIN {X 0,Y 566.855,Z 543.492,A -85,B 0,C 180,E1 -2597.697,E2 -2597.697} C_VEL
LIN {X 0,Y 566.744,Z 556.402,A -85,B 0,C 180,E1 -2598.149,E2 -2598.149} C_VEL
LIN {X 0,Y 566.594,Z 567.454,A -85,B 0,C 180,E1 -2598.671,E2 -2598.671} C_VEL
LIN {X 0,Y 566.491,Z 578.923,A -85,B 0,C 180,E1 -2599.367,E2 -2599.367} C_VEL
LIN {X 0,Y 566.332,Z 589.552,A -85,B 0,C 180,E1 -2600.176,E2 -2600.176} C_VEL
LIN {X 0,Y 566.206,Z 599.123,A -85,B 0,C 180,E1 -2601.075,E2 -2601.075} C_VEL
LIN {X 0,Y 566.111,Z 606.969,A -85,B 0,C 180,E1 -2601.973,E2 -2601.973} C_VEL
LIN {X 0,Y 566,Z 614.628,A -85,B 0,C 180,E1 -2603.048,E2 -2603.048} C_VEL
LIN {X 0,Y 566.003,Z 621.685,A -85,B 0,C 180,E1 -2604.3,E2 -2604.3} C_VEL
LIN {X 0,Y 565.933,Z 626.376,A -85,B 0,C 180,E1 -2605.371,E2 -2605.371} C_VEL
LIN {X 0,Y 565.927,Z 629.96,A -85,B 0,C 180,E1 -2606.441,E2 -2606.441} C_VEL
LIN {X 0,Y 565.878,Z 631.81,A -85,B 0,C 180,E1 -2607.153,E2 -2607.153} C_VEL
LIN {X 0,Y 565.846,Z 634.186,A -85,B 0,C 180,E1 -2608.578,E2 -2608.578} C_VEL
LIN {X 0,Y 565.839,Z 635,A -85,B 0,C 180,E1 -2610.001,E2 -2610.001} C_VEL
LIN {X 0,Y 565.846,Z 634.185,A -85,B 0,C 180,E1 -2611.424,E2 -2611.424} C_VEL
LIN {X 0,Y 565.878,Z 631.808,A -85,B 0,C 180,E1 -2612.848,E2 -2612.848} C_VEL
LIN {X 0,Y 565.926,Z 628.893,A -85,B 0,C 180,E1 -2613.917,E2 -2613.917} C_VEL
LIN {X 0,Y 565.878,Z 624.945,A -85,B 0,C 180,E1 -2614.988,E2 -2614.988} C_VEL
LIN {X 0,Y 566.002,Z 619.862,A -85,B 0,C 180,E1 -2616.059,E2 -2616.059} C_VEL
LIN {X 0,Y 566.041,Z 613.462,A -85,B 0,C 180,E1 -2617.133,E2 -2617.133} C_VEL
LIN {X 0,Y 566.133,Z 605.471,A -85,B 0,C 180,E1 -2618.209,E2 -2618.209} C_VEL
LIN {X 0,Y 566.229,Z 597.327,A -85,B 0,C 180,E1 -2619.106,E2 -2619.106} C_VEL
LIN {X 0,Y 566.343,Z 587.39,A -85,B 0,C 180,E1 -2620.006,E2 -2620.006} C_VEL
LIN {X 0,Y 566.53,Z 576.278,A -85,B 0,C 180,E1 -2620.808,E2 -2620.808} C_VEL
LIN {X 0,Y 566.614,Z 565.159,A -85,B 0,C 180,E1 -2621.448,E2 -2621.448} C_VEL
LIN {X 0,Y 566.771,Z 552.961,A -85,B 0,C 180,E1 -2621.988,E2 -2621.988} C_VEL
LIN {X 0,Y 566.909,Z 540.142,A -85,B 0,C 180,E1 -2622.394,E2 -2622.394} C_VEL
LIN {X 0,Y 566.988,Z 528.05,A -85,B 0,C 180,E1 -2622.643,E2 -2622.643} C_VEL
LIN {X 0,Y 567.038,Z 427.298,A -85,B 0,C 180,E1 -2623.933,E2 -2623.933} C_VEL
LIN {X 0,Y 566.378,Z 422.787,A -85,B 0,C 180,E1 -2624.026,E2 -2624.026} C_VEL
LIN {X 0,Y 566.592,Z 401.707,A -85,B 0,C 180,E1 -2627.109,E2 -2627.109} C_VEL
LIN {X 0,Y 566.852,Z 381.387,A -85,B 0,C 180,E1 -2630.125,E2 -2630.125} C_VEL
LIN {X 0,Y 567.053,Z 366.132,A -85,B 0,C 180,E1 -2632.403,E2 -2632.403} C_VEL
LIN {X 0,Y 566.215,Z 360.961,A -85,B 0,C 180,E1 -2633.235,E2 -2633.235} C_VEL
LIN {X 0,Y 566.22,Z 360.954,A -85,B 0,C 180,E1 -2635.749,E2 -2635.749} C_VEL
LIN {X 0,Y 566.208,Z 360.952,A -85,B 0,C 180,E1 -2638.203,E2 -2638.203} C_VEL
LIN {X 0,Y 566.205,Z 360.958,A -85,B 0,C 180,E1 -2641.078,E2 -2641.078} C_VEL
LIN {X 0,Y 566.218,Z 360.952,A -85,B 0,C 180,E1 -2643.735,E2 -2643.735} C_VEL
LIN {X 0,Y 566.206,Z 360.953,A -85,B 0,C 180,E1 -2646.57,E2 -2646.57} C_VEL
LIN {X 0,Y 566.228,Z 360.951,A -85,B 0,C 180,E1 -2649.687,E2 -2649.687} C_VEL
LIN {X 0,Y 566.207,Z 360.959,A -85,B 0,C 180,E1 -2652.918,E2 -2652.918} C_VEL
LIN {X 0,Y 566.204,Z 360.951,A -85,B 0,C 180,E1 -2656.049,E2 -2656.049} C_VEL
LIN {X 0,Y 566.209,Z 360.954,A -85,B 0,C 180,E1 -2659.215,E2 -2659.215} C_VEL
LIN {X 0,Y 566.188,Z 360.953,A -85,B 0,C 180,E1 -2661.637,E2 -2661.637} C_VEL
LIN {X 0,Y 566.167,Z 360.958,A -85,B 0,C 180,E1 -2664.308,E2 -2664.308} C_VEL
LIN {X 0,Y 566.225,Z 360.956,A -85,B 0,C 180,E1 -2666.898,E2 -2666.898} C_VEL
LIN {X 0,Y 566.185,Z 360.953,A -85,B 0,C 180,E1 -2669.407,E2 -2669.407} C_VEL
LIN {X 0,Y 566.2,Z 360.952,A -85,B 0,C 180,E1 -2671.857,E2 -2671.857} C_VEL
LIN {X 0,Y 566.215,Z 360.953,A -85,B 0,C 180,E1 -2674.251,E2 -2674.251} C_VEL
LIN {X 0,Y 566.177,Z 360.96,A -85,B 0,C 180,E1 -2676.719,E2 -2676.719} C_VEL
LIN {X 0,Y 566.218,Z 360.95,A -85,B 0,C 180,E1 -2679.663,E2 -2679.663} C_VEL
LIN {X 0,Y 566.204,Z 360.957,A -85,B 0,C 180,E1 -2682.668,E2 -2682.668} C_VEL
LIN {X 0,Y 566.239,Z 360.946,A -85,B 0,C 180,E1 -2685.627,E2 -2685.627} C_VEL
LIN {X 0,Y 566.24,Z 360.949,A -85,B 0,C 180,E1 -2688.675,E2 -2688.675} C_VEL
LIN {X 0,Y 566.232,Z 360.948,A -85,B 0,C 180,E1 -2691.434,E2 -2691.434} C_VEL
LIN {X 0,Y 566.264,Z 360.952,A -85,B 0,C 180,E1 -2694.302,E2 -2694.302} C_VEL
LIN {X 0,Y 566.287,Z 360.945,A -85,B 0,C 180,E1 -2697.866,E2 -2697.866} C_VEL
LIN {X 0,Y 566.306,Z 360.939,A -85,B 0,C 180,E1 -2700.711,E2 -2700.711} C_VEL
LIN {X 0,Y 566.277,Z 360.942,A -85,B 0,C 180,E1 -2702.846,E2 -2702.846} C_VEL
LIN {X 0,Y 566.264,Z 360.949,A -85,B 0,C 180,E1 -2705.698,E2 -2705.698} C_VEL
LIN {X 0,Y 566.233,Z 360.948,A -85,B 0,C 180,E1 -2708.566,E2 -2708.566} C_VEL
LIN {X 0,Y 566.248,Z 360.95,A -85,B 0,C 180,E1 -2711.454,E2 -2711.454} C_VEL
LIN {X 0,Y 566.24,Z 360.947,A -85,B 0,C 180,E1 -2714.507,E2 -2714.507} C_VEL
LIN {X 0,Y 566.205,Z 360.955,A -85,B 0,C 180,E1 -2717.332,E2 -2717.332} C_VEL
LIN {X 0,Y 566.218,Z 360.951,A -85,B 0,C 180,E1 -2720.337,E2 -2720.337} C_VEL
LIN {X 0,Y 566.178,Z 360.96,A -85,B 0,C 180,E1 -2723.282,E2 -2723.282} C_VEL
LIN {X 0,Y 566.22,Z 360.956,A -85,B 0,C 180,E1 -2725.749,E2 -2725.749} C_VEL
LIN {X 0,Y 566.203,Z 360.957,A -85,B 0,C 180,E1 -2727.482,E2 -2727.482} C_VEL
LIN {X 0,Y 565.517,Z 361.04,A -85,B 0,C 180,E1 -2728.076,E2 -2728.076} C_VEL
LIN {X 0,Y 562.653,Z 361.398,A -85,B 0,C 180,E1 -2729.039,E2 -2729.039} C_VEL
LIN {X 0,Y 560.249,Z 361.699,A -85,B 0,C 180,E1 -2729.815,E2 -2729.815} C_VEL
LIN {X 0,Y 559.225,Z 361.823,A -85,B 0,C 180,E1 -2730.414,E2 -2730.414} C_VEL
LIN {X 0,Y 559.145,Z 361.833,A -85,B 0,C 180,E1 -2730.617,E2 -2730.617} C_VEL
LIN {X 0,Y 559.192,Z 361.923,A -85,B 0,C 180,E1 -2732.047,E2 -2732.047} C_VEL
LIN {X 0,Y 559.57,Z 366.475,A -85,B 0,C 180,E1 -2732.902,E2 -2732.902} C_VEL
LIN {X 0,Y 559.35,Z 383.49,A -85,B 0,C 180,E1 -2735.973,E2 -2735.973} C_VEL
LIN {X 0,Y 559.222,Z 394.161,A -85,B 0,C 180,E1 -2737.867,E2 -2737.867} C_VEL
LIN {X 0,Y 560.303,Z 401.509,A -85,B 0,C 180,E1 -2737.996,E2 -2737.996} C_VEL
LIN {X 0,Y 560.025,Z 501.163,A -85,B 0,C 180,E1 -2739.295,E2 -2739.295} C_VEL
LIN {X 0,Y 559.91,Z 514.164,A -85,B 0,C 180,E1 -2739.606,E2 -2739.606} C_VEL
LIN {X 0,Y 559.774,Z 527.064,A -85,B 0,C 180,E1 -2740.072,E2 -2740.072} C_VEL
LIN {X 0,Y 559.603,Z 539.225,A -85,B 0,C 180,E1 -2740.671,E2 -2740.671} C_VEL
LIN {X 0,Y 559.45,Z 550.495,A -85,B 0,C 180,E1 -2741.386,E2 -2741.386} C_VEL
LIN {X 0,Y 559.271,Z 561.314,A -85,B 0,C 180,E1 -2742.25,E2 -2742.25} C_VEL
LIN {X 0,Y 559.139,Z 570.874,A -85,B 0,C 180,E1 -2743.195,E2 -2743.195} C_VEL
LIN {X 0,Y 559.027,Z 579.31,A -85,B 0,C 180,E1 -2744.225,E2 -2744.225} C_VEL
LIN {X 0,Y 558.926,Z 586.071,A -85,B 0,C 180,E1 -2745.238,E2 -2745.238} C_VEL
LIN {X 0,Y 558.873,Z 591.522,A -85,B 0,C 180,E1 -2746.239,E2 -2746.239} C_VEL
LIN {X 0,Y 558.84,Z 595.867,A -85,B 0,C 180,E1 -2747.225,E2 -2747.225} C_VEL
LIN {X 0,Y 558.815,Z 600.487,A -85,B 0,C 180,E1 -2748.624,E2 -2748.624} C_VEL
LIN {X 0,Y 558.768,Z 601.785,A -85,B 0,C 180,E1 -2749.152,E2 -2749.152} C_VEL
LIN {X 0,Y 558.77,Z 603.543,A -85,B 0,C 180,E1 -2750.107,E2 -2750.107} C_VEL
LIN {X 0,Y 558.733,Z 604.735,A -85,B 0,C 180,E1 -2751.249,E2 -2751.249} C_VEL
LIN {X 0,Y 558.726,Z 604.926,A -85,B 0,C 180,E1 -2752.416,E2 -2752.416} C_VEL
LIN {X 0,Y 558.729,Z 603.881,A -85,B 0,C 180,E1 -2753.758,E2 -2753.758} C_VEL
LIN {X 0,Y 558.772,Z 602.001,A -85,B 0,C 180,E1 -2754.84,E2 -2754.84} C_VEL
LIN {X 0,Y 558.82,Z 598.587,A -85,B 0,C 180,E1 -2756.104,E2 -2756.104} C_VEL
LIN {X 0,Y 558.86,Z 593.577,A -85,B 0,C 180,E1 -2757.413,E2 -2757.413} C_VEL
LIN {X 0,Y 558.917,Z 588.279,A -85,B 0,C 180,E1 -2758.472,E2 -2758.472} C_VEL
LIN {X 0,Y 558.997,Z 581.233,A -85,B 0,C 180,E1 -2759.599,E2 -2759.599} C_VEL
LIN {X 0,Y 559.114,Z 573.08,A -85,B 0,C 180,E1 -2760.644,E2 -2760.644} C_VEL
LIN {X 0,Y 559.234,Z 563.869,A -85,B 0,C 180,E1 -2761.607,E2 -2761.607} C_VEL
LIN {X 0,Y 559.431,Z 553.211,A -85,B 0,C 180,E1 -2762.504,E2 -2762.504} C_VEL
LIN {X 0,Y 559.609,Z 542.168,A -85,B 0,C 180,E1 -2763.247,E2 -2763.247} C_VEL
LIN {X 0,Y 559.717,Z 530.228,A -85,B 0,C 180,E1 -2763.879,E2 -2763.879} C_VEL
LIN {X 0,Y 559.905,Z 517.291,A -85,B 0,C 180,E1 -2764.385,E2 -2764.385} C_VEL
LIN {X 0,Y 560.039,Z 505.022,A -85,B 0,C 180,E1 -2764.719,E2 -2764.719} C_VEL
LIN {X 0,Y 560.074,Z 489.176,A -85,B 0,C 180,E1 -2764.968,E2 -2764.968} C_VEL
LIN {X 0,Y 560.251,Z 400.309,A -85,B 0,C 180,E1 -2766.111,E2 -2766.111} C_VEL
LIN {X 0,Y 559.271,Z 394.064,A -85,B 0,C 180,E1 -2766.239,E2 -2766.239} C_VEL
LIN {X 0,Y 559.427,Z 377.366,A -85,B 0,C 180,E1 -2769.212,E2 -2769.212} C_VEL
LIN {X 0,Y 559.572,Z 364.703,A -85,B 0,C 180,E1 -2771.51,E2 -2771.51} C_VEL
LIN {X 0,Y 559.223,Z 361.829,A -85,B 0,C 180,E1 -2772.066,E2 -2772.066} C_VEL
LIN {X 0,Y 559.203,Z 361.824,A -85,B 0,C 180,E1 -2775.441,E2 -2775.441} C_VEL
LIN {X 0,Y 559.212,Z 361.832,A -85,B 0,C 180,E1 -2778.604,E2 -2778.604} C_VEL
LIN {X 0,Y 559.191,Z 361.824,A -85,B 0,C 180,E1 -2781.325,E2 -2781.325} C_VEL
LIN {X 0,Y 559.229,Z 361.826,A -85,B 0,C 180,E1 -2784.229,E2 -2784.229} C_VEL
LIN {X 0,Y 559.258,Z 361.818,A -85,B 0,C 180,E1 -2787.839,E2 -2787.839} C_VEL
LIN {X 0,Y 559.277,Z 361.817,A -85,B 0,C 180,E1 -2790.719,E2 -2790.719} C_VEL
LIN {X 0,Y 559.242,Z 361.819,A -85,B 0,C 180,E1 -2792.88,E2 -2792.88} C_VEL
LIN {X 0,Y 559.23,Z 361.822,A -85,B 0,C 180,E1 -2795.769,E2 -2795.769} C_VEL
LIN {X 0,Y 559.188,Z 361.827,A -85,B 0,C 180,E1 -2798.673,E2 -2798.673} C_VEL
LIN {X 0,Y 559.208,Z 361.824,A -85,B 0,C 180,E1 -2801.599,E2 -2801.599} C_VEL
LIN {X 0,Y 559.202,Z 361.825,A -85,B 0,C 180,E1 -2804.594,E2 -2804.594} C_VEL
LIN {X 0,Y 559.164,Z 361.831,A -85,B 0,C 180,E1 -2807.556,E2 -2807.556} C_VEL
LIN {X 0,Y 559.166,Z 361.835,A -85,B 0,C 180,E1 -2809.836,E2 -2809.836} C_VEL
LIN {X 0,Y 559.141,Z 361.836,A -85,B 0,C 180,E1 -2812.152,E2 -2812.152} C_VEL
LIN {X 0,Y 559.176,Z 361.828,A -85,B 0,C 180,E1 -2815.297,E2 -2815.297} C_VEL
LIN {X 0,Y 559.188,Z 361.833,A -85,B 0,C 180,E1 -2817.71,E2 -2817.71} C_VEL
LIN {X 0,Y 559.167,Z 361.83,A -85,B 0,C 180,E1 -2820.181,E2 -2820.181} C_VEL
LIN {X 0,Y 559.173,Z 361.826,A -85,B 0,C 180,E1 -2822.713,E2 -2822.713} C_VEL
LIN {X 0,Y 559.157,Z 361.833,A -85,B 0,C 180,E1 -2825.32,E2 -2825.32} C_VEL
LIN {X 0,Y 559.131,Z 361.835,A -85,B 0,C 180,E1 -2828.016,E2 -2828.016} C_VEL
LIN {X 0,Y 559.172,Z 361.827,A -85,B 0,C 180,E1 -2830.809,E2 -2830.809} C_VEL
LIN {X 0,Y 559.157,Z 361.835,A -85,B 0,C 180,E1 -2833.731,E2 -2833.731} C_VEL
LIN {X 0,Y 559.166,Z 361.83,A -85,B 0,C 180,E1 -2836.8,E2 -2836.8} C_VEL
LIN {X 0,Y 559.232,Z 361.96,A -85,B 0,C 180,E1 -2838.102,E2 -2838.102} C_VEL
LIN {X 0,Y 559.574,Z 366.32,A -85,B 0,C 180,E1 -2838.899,E2 -2838.899} C_VEL
LIN {X 0,Y 559.396,Z 382.469,A -85,B 0,C 180,E1 -2841.792,E2 -2841.792} C_VEL
LIN {X 0,Y 559.241,Z 394.138,A -85,B 0,C 180,E1 -2843.863,E2 -2843.863} C_VEL
LIN {X 0,Y 560.294,Z 401.003,A -85,B 0,C 180,E1 -2843.989,E2 -2843.989} C_VEL
LIN {X 0,Y 560.021,Z 500.549,A -85,B 0,C 180,E1 -2845.289,E2 -2845.289} C_VEL
LIN {X 0,Y 559.969,Z 511.312,A -85,B 0,C 180,E1 -2845.531,E2 -2845.531} C_VEL
LIN {X 0,Y 559.846,Z 522.586,A -85,B 0,C 180,E1 -2845.896,E2 -2845.896} C_VEL
LIN {X 0,Y 559.663,Z 535.298,A -85,B 0,C 180,E1 -2846.459,E2 -2846.459} C_VEL
LIN {X 0,Y 559.494,Z 546.136,A -85,B 0,C 180,E1 -2847.093,E2 -2847.093} C_VEL
LIN {X 0,Y 559.36,Z 554.973,A -85,B 0,C 180,E1 -2847.725,E2 -2847.725} C_VEL
LIN {X 0,Y 559.254,Z 563.583,A -85,B 0,C 180,E1 -2848.464,E2 -2848.464} C_VEL
LIN {X 0,Y 559.148,Z 570.754,A -85,B 0,C 180,E1 -2849.19,E2 -2849.19} C_VEL
LIN {X 0,Y 559.039,Z 577.707,A -85,B 0,C 180,E1 -2850.02,E2 -2850.02} C_VEL
LIN {X 0,Y 558.958,Z 584.849,A -85,B 0,C 180,E1 -2851.048,E2 -2851.048} C_VEL
LIN {X 0,Y 558.88,Z 590.119,A -85,B 0,C 180,E1 -2851.969,E2 -2851.969} C_VEL
LIN {X 0,Y 558.85,Z 595.907,A -85,B 0,C 180,E1 -2853.235,E2 -2853.235} C_VEL
LIN {X 0,Y 558.817,Z 599.522,A -85,B 0,C 180,E1 -2854.285,E2 -2854.285} C_VEL
LIN {X 0,Y 558.758,Z 602.466,A -85,B 0,C 180,E1 -2855.476,E2 -2855.476} C_VEL
LIN {X 0,Y 558.766,Z 604.249,A -85,B 0,C 180,E1 -2856.657,E2 -2856.657} C_VEL
LIN {X 0,Y 558.741,Z 604.943,A -85,B 0,C 180,E1 -2857.83,E2 -2857.83} C_VEL
LIN {X 0,Y 558.761,Z 604.879,A -85,B 0,C 180,E1 -2858.607,E2 -2858.607} C_VEL
LIN {X 0,Y 558.758,Z 604.295,A -85,B 0,C 180,E1 -2859.379,E2 -2859.379} C_VEL
LIN {X 0,Y 558.762,Z 602.463,A -85,B 0,C 180,E1 -2860.615,E2 -2860.615} C_VEL
LIN {X 0,Y 558.816,Z 598.712,A -85,B 0,C 180,E1 -2862.054,E2 -2862.054} C_VEL
LIN {X 0,Y 558.85,Z 594.508,A -85,B 0,C 180,E1 -2863.187,E2 -2863.187} C_VEL
LIN {X 0,Y 558.888,Z 589.105,A -85,B 0,C 180,E1 -2864.314,E2 -2864.314} C_VEL
LIN {X 0,Y 558.986,Z 582.02,A -85,B 0,C 180,E1 -2865.484,E2 -2865.484} C_VEL
LIN {X 0,Y 559.074,Z 573.85,A -85,B 0,C 180,E1 -2866.552,E2 -2866.552} C_VEL
LIN {X 0,Y 559.225,Z 565.124,A -85,B 0,C 180,E1 -2867.479,E2 -2867.479} C_VEL
LIN {X 0,Y 559.333,Z 556.791,A -85,B 0,C 180,E1 -2868.218,E2 -2868.218} C_VEL
LIN {X 0,Y 559.471,Z 547.119,A -85,B 0,C 180,E1 -2868.931,E2 -2868.931} C_VEL
LIN {X 0,Y 559.689,Z 535.867,A -85,B 0,C 180,E1 -2869.601,E2 -2869.601} C_VEL
LIN {X 0,Y 559.816,Z 522.529,A -85,B 0,C 180,E1 -2870.197,E2 -2870.197} C_VEL
LIN {X 0,Y 559.912,Z 511.209,A -85,B 0,C 180,E1 -2870.563,E2 -2870.563} C_VEL
LIN {X 0,Y 560.036,Z 501,A -85,B 0,C 180,E1 -2870.793,E2 -2870.793} C_VEL
LIN {X 0,Y 560.183,Z 440.683,A -85,B 0,C 180,E1 -2871.591,E2 -2871.591} C_VEL
LIN {X 0,Y 560.176,Z 399.779,A -85,B 0,C 180,E1 -2872.12,E2 -2872.12} C_VEL
LIN {X 0,Y 559.255,Z 394.116,A -85,B 0,C 180,E1 -2872.23,E2 -2872.23} C_VEL
LIN {X 0,Y 559.409,Z 377.796,A -85,B 0,C 180,E1 -2875.135,E2 -2875.135} C_VEL
LIN {X 0,Y 559.507,Z 364.715,A -85,B 0,C 180,E1 -2877.48,E2 -2877.48} C_VEL
LIN {X 0,Y 559.232,Z 361.826,A -85,B 0,C 180,E1 -2878.019,E2 -2878.019} C_VEL
LIN {X 0,Y 559.269,Z 361.824,A -85,B 0,C 180,E1 -2880.72,E2 -2880.72} C_VEL
LIN {X 0,Y 559.237,Z 361.825,A -85,B 0,C 180,E1 -2882.881,E2 -2882.881} C_VEL
LIN {X 0,Y 559.222,Z 361.823,A -85,B 0,C 180,E1 -2885.77,E2 -2885.77} C_VEL
LIN {X 0,Y 559.194,Z 361.829,A -85,B 0,C 180,E1 -2888.674,E2 -2888.674} C_VEL
LIN {X 0,Y 559.199,Z 361.826,A -85,B 0,C 180,E1 -2891.601,E2 -2891.601} C_VEL
LIN {X 0,Y 559.188,Z 361.829,A -85,B 0,C 180,E1 -2894.596,E2 -2894.596} C_VEL
LIN {X 0,Y 559.156,Z 361.832,A -85,B 0,C 180,E1 -2897.557,E2 -2897.557} C_VEL
LIN {X 0,Y 559.166,Z 361.835,A -85,B 0,C 180,E1 -2899.838,E2 -2899.838} C_VEL
LIN {X 0,Y 559.148,Z 361.836,A -85,B 0,C 180,E1 -2902.153,E2 -2902.153} C_VEL
LIN {X 0,Y 559.158,Z 361.83,A -85,B 0,C 180,E1 -2904.505,E2 -2904.505} C_VEL
LIN {X 0,Y 559.172,Z 361.827,A -85,B 0,C 180,E1 -2906.902,E2 -2906.902} C_VEL
LIN {X 0,Y 559.181,Z 361.833,A -85,B 0,C 180,E1 -2909.866,E2 -2909.866} C_VEL
LIN {X 0,Y 559.168,Z 361.828,A -85,B 0,C 180,E1 -2912.715,E2 -2912.715} C_VEL
LIN {X 0,Y 559.15,Z 361.836,A -85,B 0,C 180,E1 -2915.323,E2 -2915.323} C_VEL
LIN {X 0,Y 559.128,Z 361.835,A -85,B 0,C 180,E1 -2918.018,E2 -2918.018} C_VEL
LIN {X 0,Y 559.169,Z 361.829,A -85,B 0,C 180,E1 -2920.811,E2 -2920.811} C_VEL
LIN {X 0,Y 559.158,Z 361.832,A -85,B 0,C 180,E1 -2923.732,E2 -2923.732} C_VEL
LIN {X 0,Y 559.14,Z 361.835,A -85,B 0,C 180,E1 -2926.804,E2 -2926.804} C_VEL
LIN {X 0,Y 559.171,Z 361.836,A -85,B 0,C 180,E1 -2929.191,E2 -2929.191} C_VEL
LIN {X 0,Y 559.131,Z 361.832,A -85,B 0,C 180,E1 -2931.984,E2 -2931.984} C_VEL
LIN {X 0,Y 559.158,Z 361.836,A -85,B 0,C 180,E1 -2934.784,E2 -2934.784} C_VEL
LIN {X 0,Y 559.171,Z 361.83,A -85,B 0,C 180,E1 -2937.362,E2 -2937.362} C_VEL
LIN {X 0,Y 559.187,Z 361.827,A -85,B 0,C 180,E1 -2940.136,E2 -2940.136} C_VEL
LIN {X 0,Y 559.181,Z 361.83,A -85,B 0,C 180,E1 -2943.171,E2 -2943.171} C_VEL
LIN {X 0,Y 559.156,Z 361.832,A -85,B 0,C 180,E1 -2945.496,E2 -2945.496} C_VEL
LIN {X 0,Y 559.176,Z 362.045,A -85,B 0,C 180,E1 -2946.651,E2 -2946.651} C_VEL
LIN {X 0,Y 560.111,Z 367.33,A -85,B 0,C 180,E1 -2947.5,E2 -2947.5} C_VEL
LIN {X 0,Y 559.85,Z 386.677,A -85,B 0,C 180,E1 -2950.423,E2 -2950.423} C_VEL
LIN {X 0,Y 559.578,Z 405.327,A -85,B 0,C 180,E1 -2953.211,E2 -2953.211} C_VEL
LIN {X 0,Y 559.378,Z 422.8,A -85,B 0,C 180,E1 -2955.796,E2 -2955.796} C_VEL
LIN {X 0,Y 560.306,Z 430.381,A -85,B 0,C 180,E1 -2955.936,E2 -2955.936} C_VEL
LIN {X 0,Y 560.081,Z 530.999,A -85,B 0,C 180,E1 -2957.247,E2 -2957.247} C_VEL
LIN {X 0,Y 559.917,Z 543.491,A -85,B 0,C 180,E1 -2957.542,E2 -2957.542} C_VEL
LIN {X 0,Y 559.805,Z 556.403,A -85,B 0,C 180,E1 -2958,E2 -2958} C_VEL
LIN {X 0,Y 559.617,Z 568.508,A -85,B 0,C 180,E1 -2958.585,E2 -2958.585} C_VEL
LIN {X 0,Y 559.461,Z 580.212,A -85,B 0,C 180,E1 -2959.323,E2 -2959.323} C_VEL
LIN {X 0,Y 559.301,Z 590.615,A -85,B 0,C 180,E1 -2960.143,E2 -2960.143} C_VEL
LIN {X 0,Y 559.161,Z 599.123,A -85,B 0,C 180,E1 -2960.962,E2 -2960.962} C_VEL
LIN {X 0,Y 559.049,Z 606.969,A -85,B 0,C 180,E1 -2961.871,E2 -2961.871} C_VEL
LIN {X 0,Y 558.942,Z 614.628,A -85,B 0,C 180,E1 -2962.959,E2 -2962.959} C_VEL
LIN {X 0,Y 558.935,Z 621.685,A -85,B 0,C 180,E1 -2964.228,E2 -2964.228} C_VEL
LIN {X 0,Y 558.827,Z 626.376,A -85,B 0,C 180,E1 -2965.312,E2 -2965.312} C_VEL
LIN {X 0,Y 558.836,Z 629.961,A -85,B 0,C 180,E1 -2966.396,E2 -2966.396} C_VEL
LIN {X 0,Y 558.799,Z 631.81,A -85,B 0,C 180,E1 -2967.117,E2 -2967.117} C_VEL
LIN {X 0,Y 558.745,Z 634.185,A -85,B 0,C 180,E1 -2968.559,E2 -2968.559} C_VEL
LIN {X 0,Y 558.74,Z 635,A -85,B 0,C 180,E1 -2970.001,E2 -2970.001} C_VEL
LIN {X 0,Y 558.745,Z 634.184,A -85,B 0,C 180,E1 -2971.442,E2 -2971.442} C_VEL
LIN {X 0,Y 558.799,Z 631.808,A -85,B 0,C 180,E1 -2972.885,E2 -2972.885} C_VEL
LIN {X 0,Y 558.844,Z 628.893,A -85,B 0,C 180,E1 -2973.967,E2 -2973.967} C_VEL
LIN {X 0,Y 558.799,Z 624.945,A -85,B 0,C 180,E1 -2975.052,E2 -2975.052} C_VEL
LIN {X 0,Y 558.921,Z 619.862,A -85,B 0,C 180,E1 -2976.136,E2 -2976.136} C_VEL
LIN {X 0,Y 558.978,Z 613.462,A -85,B 0,C 180,E1 -2977.224,E2 -2977.224} C_VEL
LIN {X 0,Y 559.097,Z 605.471,A -85,B 0,C 180,E1 -2978.313,E2 -2978.313} C_VEL
LIN {X 0,Y 559.185,Z 597.326,A -85,B 0,C 180,E1 -2979.222,E2 -2979.222} C_VEL
LIN {X 0,Y 559.352,Z 587.389,A -85,B 0,C 180,E1 -2980.132,E2 -2980.132} C_VEL
LIN {X 0,Y 559.543,Z 576.386,A -85,B 0,C 180,E1 -2980.938,E2 -2980.938} C_VEL
LIN {X 0,Y 559.673,Z 564.443,A -85,B 0,C 180,E1 -2981.629,E2 -2981.629} C_VEL
LIN {X 0,Y 559.83,Z 551.744,A -85,B 0,C 180,E1 -2982.185,E2 -2982.185} C_VEL
LIN {X 0,Y 560.001,Z 538.312,A -85,B 0,C 180,E1 -2982.596,E2 -2982.596} C_VEL
LIN {X 0,Y 560.094,Z 526.546,A -85,B 0,C 180,E1 -2982.824,E2 -2982.824} C_VEL
LIN {X 0,Y 560.194,Z 428.243,A -85,B 0,C 180,E1 -2984.095,E2 -2984.095} C_VEL
LIN {X 0,Y 559.374,Z 422.787,A -85,B 0,C 180,E1 -2984.206,E2 -2984.206} C_VEL
LIN {X 0,Y 559.627,Z 401.482,A -85,B 0,C 180,E1 -2987.362,E2 -2987.362} C_VEL
LIN {X 0,Y 559.927,Z 381.26,A -85,B 0,C 180,E1 -2990.385,E2 -2990.385} C_VEL
LIN {X 0,Y 560.075,Z 367.216,A -85,B 0,C 180,E1 -2992.503,E2 -2992.503} C_VEL
LIN {X 0,Y 559.158,Z 361.84,A -85,B 0,C 180,E1 -2993.394,E2 -2993.394} C_VEL
LIN {X 0,Y 559.187,Z 361.827,A -85,B 0,C 180,E1 -2996.098,E2 -2996.098} C_VEL
LIN {X 0,Y 559.169,Z 361.83,A -85,B 0,C 180,E1 -2998.53,E2 -2998.53} C_VEL
LIN {X 0,Y 559.159,Z 361.839,A -85,B 0,C 180,E1 -3001.275,E2 -3001.275} C_VEL
LIN {X 0,Y 559.173,Z 361.828,A -85,B 0,C 180,E1 -3003.95,E2 -3003.95} C_VEL
LIN {X 0,Y 559.147,Z 361.84,A -85,B 0,C 180,E1 -3007.109,E2 -3007.109} C_VEL
LIN {X 0,Y 559.171,Z 361.828,A -85,B 0,C 180,E1 -3009.943,E2 -3009.943} C_VEL
LIN {X 0,Y 559.163,Z 361.834,A -85,B 0,C 180,E1 -3012.744,E2 -3012.744} C_VEL
LIN {X 0,Y 559.159,Z 361.829,A -85,B 0,C 180,E1 -3015.761,E2 -3015.761} C_VEL
LIN {X 0,Y 559.169,Z 361.828,A -85,B 0,C 180,E1 -3018.23,E2 -3018.23} C_VEL
LIN {X 0,Y 559.178,Z 361.831,A -85,B 0,C 180,E1 -3021.192,E2 -3021.192} C_VEL
LIN {X 0,Y 559.143,Z 361.83,A -85,B 0,C 180,E1 -3023.789,E2 -3023.789} C_VEL
LIN {X 0,Y 559.168,Z 361.831,A -85,B 0,C 180,E1 -3026.425,E2 -3026.425} C_VEL
LIN {X 0,Y 559.16,Z 361.832,A -85,B 0,C 180,E1 -3028.981,E2 -3028.981} C_VEL
LIN {X 0,Y 559.174,Z 361.827,A -85,B 0,C 180,E1 -3031.619,E2 -3031.619} C_VEL
LIN {X 0,Y 559.181,Z 361.834,A -85,B 0,C 180,E1 -3034.702,E2 -3034.702} C_VEL
LIN {X 0,Y 559.147,Z 361.83,A -85,B 0,C 180,E1 -3037.847,E2 -3037.847} C_VEL
LIN {X 0,Y 559.199,Z 361.831,A -85,B 0,C 180,E1 -3040.494,E2 -3040.494} C_VEL
LIN {X 0,Y 559.186,Z 361.826,A -85,B 0,C 180,E1 -3043.198,E2 -3043.198} C_VEL
LIN {X 0,Y 559.175,Z 361.832,A -85,B 0,C 180,E1 -3046.184,E2 -3046.184} C_VEL
LIN {X 0,Y 559.2,Z 361.822,A -85,B 0,C 180,E1 -3049.134,E2 -3049.134} C_VEL
LIN {X 0,Y 559.209,Z 361.829,A -85,B 0,C 180,E1 -3052.054,E2 -3052.054} C_VEL
LIN {X 0,Y 559.258,Z 361.817,A -85,B 0,C 180,E1 -3054.953,E2 -3054.953} C_VEL
LIN {X 0,Y 559.258,Z 361.82,A -85,B 0,C 180,E1 -3057.839,E2 -3057.839} C_VEL
LIN {X 0,Y 559.276,Z 361.814,A -85,B 0,C 180,E1 -3060.72,E2 -3060.72} C_VEL
LIN {X 0,Y 559.244,Z 361.818,A -85,B 0,C 180,E1 -3062.881,E2 -3062.881} C_VEL
LIN {X 0,Y 559.234,Z 361.826,A -85,B 0,C 180,E1 -3065.77,E2 -3065.77} C_VEL
LIN {X 0,Y 559.192,Z 361.825,A -85,B 0,C 180,E1 -3068.674,E2 -3068.674} C_VEL
LIN {X 0,Y 559.212,Z 361.828,A -85,B 0,C 180,E1 -3071.6,E2 -3071.6} C_VEL
LIN {X 0,Y 559.206,Z 361.823,A -85,B 0,C 180,E1 -3074.596,E2 -3074.596} C_VEL
LIN {X 0,Y 559.164,Z 361.836,A -85,B 0,C 180,E1 -3077.557,E2 -3077.557} C_VEL
LIN {X 0,Y 559.176,Z 361.834,A -85,B 0,C 180,E1 -3079.837,E2 -3079.837} C_VEL
LIN {X 0,Y 559.148,Z 361.833,A -85,B 0,C 180,E1 -3082.153,E2 -3082.153} C_VEL
LIN {X 0,Y 559.182,Z 361.832,A -85,B 0,C 180,E1 -3085.298,E2 -3085.298} C_VEL
LIN {X 0,Y 559.153,Z 361.837,A -85,B 0,C 180,E1 -3087.714,E2 -3087.714} C_VEL
LIN {X 0,Y 559.145,Z 361.833,A -85,B 0,C 180,E1 -3090.617,E2 -3090.617} C_VEL
LIN {X 0,Y 558.527,Z 361.988,A -85,B 0,C 180,E1 -3091.024,E2 -3091.024} C_VEL
LIN {X 0,Y 555.904,Z 362.925,A -85,B 0,C 180,E1 -3091.661,E2 -3091.661} C_VEL
LIN {X 0,Y 553.258,Z 364.866,A -85,B 0,C 180,E1 -3092.276,E2 -3092.276} C_VEL
LIN {X 0,Y 552.609,Z 366.609,A -85,B 0,C 180,E1 -3092.647,E2 -3092.647} C_VEL
LIN {X 0,Y 552.35,Z 383.868,A -85,B 0,C 180,E1 -3095.824,E2 -3095.824} C_VEL
LIN {X 0,Y 552.217,Z 394.124,A -85,B 0,C 180,E1 -3097.676,E2 -3097.676} C_VEL
LIN {X 0,Y 553.437,Z 402.175,A -85,B 0,C 180,E1 -3097.826,E2 -3097.826} C_VEL
LIN {X 0,Y 553.107,Z 501.209,A -85,B 0,C 180,E1 -3099.134,E2 -3099.134} C_VEL
LIN {X 0,Y 552.979,Z 514.407,A -85,B 0,C 180,E1 -3099.455,E2 -3099.455} C_VEL
LIN {X 0,Y 552.805,Z 527.594,A -85,B 0,C 180,E1 -3099.943,E2 -3099.943} C_VEL
LIN {X 0,Y 552.618,Z 539.77,A -85,B 0,C 180,E1 -3100.556,E2 -3100.556} C_VEL
LIN {X 0,Y 552.433,Z 551.134,A -85,B 0,C 180,E1 -3101.296,E2 -3101.296} C_VEL
LIN {X 0,Y 552.241,Z 561.802,A -85,B 0,C 180,E1 -3102.169,E2 -3102.169} C_VEL
LIN {X 0,Y 552.082,Z 571.715,A -85,B 0,C 180,E1 -3103.176,E2 -3103.176} C_VEL
LIN {X 0,Y 551.959,Z 579.822,A -85,B 0,C 180,E1 -3104.197,E2 -3104.197} C_VEL
LIN {X 0,Y 551.838,Z 586.831,A -85,B 0,C 180,E1 -3105.28,E2 -3105.28} C_VEL
LIN {X 0,Y 551.787,Z 593.332,A -85,B 0,C 180,E1 -3106.552,E2 -3106.552} C_VEL
LIN {X 0,Y 551.752,Z 597.574,A -85,B 0,C 180,E1 -3107.628,E2 -3107.628} C_VEL
LIN {X 0,Y 551.711,Z 600.857,A -85,B 0,C 180,E1 -3108.727,E2 -3108.727} C_VEL
LIN {X 0,Y 551.656,Z 603.2,A -85,B 0,C 180,E1 -3109.853,E2 -3109.853} C_VEL
LIN {X 0,Y 551.643,Z 604.583,A -85,B 0,C 180,E1 -3111.001,E2 -3111.001} C_VEL
LIN {X 0,Y 551.622,Z 604.952,A -85,B 0,C 180,E1 -3112.298,E2 -3112.298} C_VEL
LIN {X 0,Y 551.649,Z 604.315,A -85,B 0,C 180,E1 -3113.381,E2 -3113.381} C_VEL
LIN {X 0,Y 551.682,Z 602.503,A -85,B 0,C 180,E1 -3114.619,E2 -3114.619} C_VEL
LIN {X 0,Y 551.721,Z 599.349,A -85,B 0,C 180,E1 -3115.91,E2 -3115.91} C_VEL
LIN {X 0,Y 551.758,Z 594.733,A -85,B 0,C 180,E1 -3117.212,E2 -3117.212} C_VEL
LIN {X 0,Y 551.847,Z 588.453,A -85,B 0,C 180,E1 -3118.523,E2 -3118.523} C_VEL
LIN {X 0,Y 551.952,Z 581.145,A -85,B 0,C 180,E1 -3119.708,E2 -3119.708} C_VEL
LIN {X 0,Y 552.081,Z 572.171,A -85,B 0,C 180,E1 -3120.861,E2 -3120.861} C_VEL
LIN {X 0,Y 552.211,Z 563.661,A -85,B 0,C 180,E1 -3121.75,E2 -3121.75} C_VEL
LIN {X 0,Y 552.442,Z 553.178,A -85,B 0,C 180,E1 -3122.64,E2 -3122.64} C_VEL
LIN {X 0,Y 552.626,Z 542.354,A -85,B 0,C 180,E1 -3123.379,E2 -3123.379} C_VEL
LIN {X 0,Y 552.787,Z 530.138,A -85,B 0,C 180,E1 -3124.034,E2 -3124.034} C_VEL
LIN {X 0,Y 552.96,Z 517.296,A -85,B 0,C 180,E1 -3124.542,E2 -3124.542} C_VEL
LIN {X 0,Y 553.126,Z 504.899,A -85,B 0,C 180,E1 -3124.883,E2 -3124.883} C_VEL
LIN {X 0,Y 553.157,Z 488.946,A -85,B 0,C 180,E1 -3125.135,E2 -3125.135} C_VEL
LIN {X 0,Y 553.268,Z 400.586,A -85,B 0,C 180,E1 -3126.289,E2 -3126.289} C_VEL
LIN {X 0,Y 552.237,Z 394.177,A -85,B 0,C 180,E1 -3126.404,E2 -3126.404} C_VEL
LIN {X 0,Y 552.463,Z 376.983,A -85,B 0,C 180,E1 -3129.522,E2 -3129.522} C_VEL
LIN {X 0,Y 552.62,Z 366.49,A -85,B 0,C 180,E1 -3131.461,E2 -3131.461} C_VEL
LIN {X 0,Y 552.172,Z 362.708,A -85,B 0,C 180,E1 -3132.213,E2 -3132.213} C_VEL
LIN {X 0,Y 552.164,Z 362.702,A -85,B 0,C 180,E1 -3135.316,E2 -3135.316} C_VEL
LIN {X 0,Y 552.182,Z 362.707,A -85,B 0,C 180,E1 -3138.533,E2 -3138.533} C_VEL
LIN {X 0,Y 552.163,Z 362.701,A -85,B 0,C 180,E1 -3141.214,E2 -3141.214} C_VEL
LIN {X 0,Y 552.198,Z 362.7,A -85,B 0,C 180,E1 -3144.155,E2 -3144.155} C_VEL
LIN {X 0,Y 552.208,Z 362.695,A -85,B 0,C 180,E1 -3147.081,E2 -3147.081} C_VEL
LIN {X 0,Y 552.237,Z 362.695,A -85,B 0,C 180,E1 -3149.999,E2 -3149.999} C_VEL
LIN {X 0,Y 552.208,Z 362.695,A -85,B 0,C 180,E1 -3152.917,E2 -3152.917} C_VEL
LIN {X 0,Y 552.201,Z 362.699,A -85,B 0,C 180,E1 -3155.843,E2 -3155.843} C_VEL
LIN {X 0,Y 552.156,Z 362.702,A -85,B 0,C 180,E1 -3158.785,E2 -3158.785} C_VEL
LIN {X 0,Y 552.166,Z 362.703,A -85,B 0,C 180,E1 -3161.749,E2 -3161.749} C_VEL
LIN {X 0,Y 552.139,Z 362.704,A -85,B 0,C 180,E1 -3164.747,E2 -3164.747} C_VEL
LIN {X 0,Y 552.114,Z 362.712,A -85,B 0,C 180,E1 -3167.787,E2 -3167.787} C_VEL
LIN {X 0,Y 552.127,Z 362.711,A -85,B 0,C 180,E1 -3170.1,E2 -3170.1} C_VEL
LIN {X 0,Y 552.092,Z 362.71,A -85,B 0,C 180,E1 -3172.45,E2 -3172.45} C_VEL
LIN {X 0,Y 552.155,Z 362.703,A -85,B 0,C 180,E1 -3175.349,E2 -3175.349} C_VEL
LIN {X 0,Y 552.122,Z 362.71,A -85,B 0,C 180,E1 -3178.096,E2 -3178.096} C_VEL
LIN {X 0,Y 552.112,Z 362.706,A -85,B 0,C 180,E1 -3180.607,E2 -3180.607} C_VEL
LIN {X 0,Y 552.121,Z 362.707,A -85,B 0,C 180,E1 -3183.184,E2 -3183.184} C_VEL
LIN {X 0,Y 552.111,Z 362.713,A -85,B 0,C 180,E1 -3185.84,E2 -3185.84} C_VEL
LIN {X 0,Y 552.122,Z 362.707,A -85,B 0,C 180,E1 -3189.061,E2 -3189.061} C_VEL
LIN {X 0,Y 552.136,Z 362.711,A -85,B 0,C 180,E1 -3191.443,E2 -3191.443} C_VEL
LIN {X 0,Y 552.091,Z 362.71,A -85,B 0,C 180,E1 -3194.531,E2 -3194.531} C_VEL
LIN {X 0,Y 552.129,Z 362.713,A -85,B 0,C 180,E1 -3197.583,E2 -3197.583} C_VEL
LIN {X 0,Y 552.182,Z 362.802,A -85,B 0,C 180,E1 -3198.015,E2 -3198.015} C_VEL
LIN {X 0,Y 552.56,Z 367.329,A -85,B 0,C 180,E1 -3198.854,E2 -3198.854} C_VEL
LIN {X 0,Y 552.377,Z 383.673,A -85,B 0,C 180,E1 -3201.792,E2 -3201.792} C_VEL
LIN {X 0,Y 552.227,Z 394.144,A -85,B 0,C 180,E1 -3203.68,E2 -3203.68} C_VEL
LIN {X 0,Y 553.406,Z 401.161,A -85,B 0,C 180,E1 -3203.812,E2 -3203.812} C_VEL
LIN {X 0,Y 553.102,Z 500.366,A -85,B 0,C 180,E1 -3205.124,E2 -3205.124} C_VEL
LIN {X 0,Y 552.998,Z 510.635,A -85,B 0,C 180,E1 -3205.353,E2 -3205.353} C_VEL
LIN {X 0,Y 552.891,Z 520.629,A -85,B 0,C 180,E1 -3205.67,E2 -3205.67} C_VEL
LIN {X 0,Y 552.746,Z 530.745,A -85,B 0,C 180,E1 -3206.092,E2 -3206.092} C_VEL
LIN {X 0,Y 552.601,Z 540.91,A -85,B 0,C 180,E1 -3206.629,E2 -3206.629} C_VEL
LIN {X 0,Y 552.401,Z 552.65,A -85,B 0,C 180,E1 -3207.407,E2 -3207.407} C_VEL
LIN {X 0,Y 552.217,Z 562.82,A -85,B 0,C 180,E1 -3208.267,E2 -3208.267} C_VEL
LIN {X 0,Y 552.13,Z 569.793,A -85,B 0,C 180,E1 -3208.968,E2 -3208.968} C_VEL
LIN {X 0,Y 552.022,Z 576.179,A -85,B 0,C 180,E1 -3209.713,E2 -3209.713} C_VEL
LIN {X 0,Y 551.88,Z 582.862,A -85,B 0,C 180,E1 -3210.641,E2 -3210.641} C_VEL
LIN {X 0,Y 551.804,Z 589.051,A -85,B 0,C 180,E1 -3211.687,E2 -3211.687} C_VEL
LIN {X 0,Y 551.771,Z 593.954,A -85,B 0,C 180,E1 -3212.707,E2 -3212.707} C_VEL
LIN {X 0,Y 551.743,Z 598.527,A -85,B 0,C 180,E1 -3213.931,E2 -3213.931} C_VEL
LIN {X 0,Y 551.68,Z 601.808,A -85,B 0,C 180,E1 -3215.14,E2 -3215.14} C_VEL
LIN {X 0,Y 551.663,Z 604.132,A -85,B 0,C 180,E1 -3216.524,E2 -3216.524} C_VEL
LIN {X 0,Y 551.648,Z 604.9,A -85,B 0,C 180,E1 -3217.53,E2 -3217.53} C_VEL
LIN {X 0,Y 551.661,Z 604.929,A -85,B 0,C 180,E1 -3218.431,E2 -3218.431} C_VEL
LIN {X 0,Y 551.65,Z 603.717,A -85,B 0,C 180,E1 -3219.88,E2 -3219.88} C_VEL
LIN {X 0,Y 551.677,Z 602.449,A -85,B 0,C 180,E1 -3220.657,E2 -3220.657} C_VEL
LIN {X 0,Y 551.708,Z 599.638,A -85,B 0,C 180,E1 -3221.814,E2 -3221.814} C_VEL
LIN {X 0,Y 551.759,Z 595.712,A -85,B 0,C 180,E1 -3222.965,E2 -3222.965} C_VEL
LIN {X 0,Y 551.778,Z 590.588,A -85,B 0,C 180,E1 -3224.107,E2 -3224.107} C_VEL
LIN {X 0,Y 551.861,Z 585.322,A -85,B 0,C 180,E1 -3225.055,E2 -3225.055} C_VEL
LIN {X 0,Y 551.954,Z 578.987,A -85,B 0,C 180,E1 -3226,E2 -3226} C_VEL
LIN {X 0,Y 552.084,Z 571.39,A -85,B 0,C 180,E1 -3226.941,E2 -3226.941} C_VEL
LIN {X 0,Y 552.211,Z 564.177,A -85,B 0,C 180,E1 -3227.691,E2 -3227.691} C_VEL
LIN {X 0,Y 552.355,Z 555.716,A -85,B 0,C 180,E1 -3228.436,E2 -3228.436} C_VEL
LIN {X 0,Y 552.516,Z 545.422,A -85,B 0,C 180,E1 -3229.186,E2 -3229.186} C_VEL
LIN {X 0,Y 552.76,Z 534.131,A -85,B 0,C 180,E1 -3229.839,E2 -3229.839} C_VEL
LIN {X 0,Y 552.861,Z 522.58,A -85,B 0,C 180,E1 -3230.349,E2 -3230.349} C_VEL
LIN {X 0,Y 552.999,Z 511.226,A -85,B 0,C 180,E1 -3230.721,E2 -3230.721} C_VEL
LIN {X 0,Y 553.115,Z 501.057,A -85,B 0,C 180,E1 -3230.953,E2 -3230.953} C_VEL
LIN {X 0,Y 553.245,Z 453.251,A -85,B 0,C 180,E1 -3231.6,E2 -3231.6} C_VEL
LIN {X 0,Y 553.357,Z 401.003,A -85,B 0,C 180,E1 -3232.281,E2 -3232.281} C_VEL
LIN {X 0,Y 552.237,Z 394.065,A -85,B 0,C 180,E1 -3232.423,E2 -3232.423} C_VEL
LIN {X 0,Y 552.394,Z 378.274,A -85,B 0,C 180,E1 -3235.256,E2 -3235.256} C_VEL
LIN {X 0,Y 552.506,Z 366.147,A -85,B 0,C 180,E1 -3237.448,E2 -3237.448} C_VEL
LIN {X 0,Y 552.196,Z 362.703,A -85,B 0,C 180,E1 -3238.085,E2 -3238.085} C_VEL
LIN {X 0,Y 552.239,Z 362.699,A -85,B 0,C 180,E1 -3240.729,E2 -3240.729} C_VEL
LIN {X 0,Y 552.203,Z 362.701,A -85,B 0,C 180,E1 -3242.918,E2 -3242.918} C_VEL
LIN {X 0,Y 552.192,Z 362.7,A -85,B 0,C 180,E1 -3245.844,E2 -3245.844} C_VEL
LIN {X 0,Y 552.162,Z 362.704,A -85,B 0,C 180,E1 -3248.786,E2 -3248.786} C_VEL
LIN {X 0,Y 552.154,Z 362.705,A -85,B 0,C 180,E1 -3251.751,E2 -3251.751} C_VEL
LIN {X 0,Y 552.127,Z 362.707,A -85,B 0,C 180,E1 -3254.749,E2 -3254.749} C_VEL
LIN {X 0,Y 552.107,Z 362.713,A -85,B 0,C 180,E1 -3257.789,E2 -3257.789} C_VEL
LIN {X 0,Y 552.125,Z 362.713,A -85,B 0,C 180,E1 -3260.101,E2 -3260.101} C_VEL
LIN {X 0,Y 552.107,Z 362.709,A -85,B 0,C 180,E1 -3262.45,E2 -3262.45} C_VEL
LIN {X 0,Y 552.153,Z 362.704,A -85,B 0,C 180,E1 -3265.353,E2 -3265.353} C_VEL
LIN {X 0,Y 552.119,Z 362.71,A -85,B 0,C 180,E1 -3268.098,E2 -3268.098} C_VEL
LIN {X 0,Y 552.107,Z 362.708,A -85,B 0,C 180,E1 -3270.609,E2 -3270.609} C_VEL
LIN {X 0,Y 552.121,Z 362.709,A -85,B 0,C 180,E1 -3273.186,E2 -3273.186} C_VEL
LIN {X 0,Y 552.105,Z 362.712,A -85,B 0,C 180,E1 -3275.842,E2 -3275.842} C_VEL
LIN {X 0,Y 552.118,Z 362.71,A -85,B 0,C 180,E1 -3279.063,E2 -3279.063} C_VEL
LIN {X 0,Y 552.133,Z 362.712,A -85,B 0,C 180,E1 -3281.445,E2 -3281.445} C_VEL
LIN {X 0,Y 552.09,Z 362.71,A -85,B 0,C 180,E1 -3284.533,E2 -3284.533} C_VEL
LIN {X 0,Y 552.125,Z 362.708,A -85,B 0,C 180,E1 -3287.585,E2 -3287.585} C_VEL
LIN {X 0,Y 552.13,Z 362.706,A -85,B 0,C 180,E1 -3290.474,E2 -3290.474} C_VEL
LIN {X 0,Y 552.111,Z 362.711,A -85,B 0,C 180,E1 -3293.317,E2 -3293.317} C_VEL
LIN {X 0,Y 552.129,Z 362.705,A -85,B 0,C 180,E1 -3295.941,E2 -3295.941} C_VEL
LIN {X 0,Y 552.115,Z 362.711,A -85,B 0,C 180,E1 -3298.542,E2 -3298.542} C_VEL
LIN {X 0,Y 552.124,Z 362.707,A -85,B 0,C 180,E1 -3301.439,E2 -3301.439} C_VEL
LIN {X 0,Y 552.136,Z 362.71,A -85,B 0,C 180,E1 -3304.357,E2 -3304.357} C_VEL
LIN {X 0,Y 552.138,Z 362.748,A -85,B 0,C 180,E1 -3306.467,E2 -3306.467} C_VEL
LIN {X 0,Y 553.163,Z 368.47,A -85,B 0,C 180,E1 -3307.399,E2 -3307.399} C_VEL
LIN {X 0,Y 552.889,Z 386.513,A -85,B 0,C 180,E1 -3310.161,E2 -3310.161} C_VEL
LIN {X 0,Y 552.594,Z 405.301,A -85,B 0,C 180,E1 -3312.992,E2 -3312.992} C_VEL
LIN {X 0,Y 552.366,Z 422.897,A -85,B 0,C 180,E1 -3315.627,E2 -3315.627} C_VEL
LIN {X 0,Y 553.42,Z 430.883,A -85,B 0,C 180,E1 -3315.764,E2 -3315.764} C_VEL
LIN {X 0,Y 553.167,Z 530.999,A -85,B 0,C 180,E1 -3317.085,E2 -3317.085} C_VEL
LIN {X 0,Y 552.993,Z 544.252,A -85,B 0,C 180,E1 -3317.407,E2 -3317.407} C_VEL
LIN {X 0,Y 552.844,Z 556.396,A -85,B 0,C 180,E1 -3317.846,E2 -3317.846} C_VEL
LIN {X 0,Y 552.641,Z 567.307,A -85,B 0,C 180,E1 -3318.373,E2 -3318.373} C_VEL
LIN {X 0,Y 552.519,Z 578.919,A -85,B 0,C 180,E1 -3319.094,E2 -3319.094} C_VEL
LIN {X 0,Y 552.293,Z 589.55,A -85,B 0,C 180,E1 -3319.924,E2 -3319.924} C_VEL
LIN {X 0,Y 552.125,Z 599.123,A -85,B 0,C 180,E1 -3320.846,E2 -3320.846} C_VEL
LIN {X 0,Y 552.012,Z 606.969,A -85,B 0,C 180,E1 -3321.766,E2 -3321.766} C_VEL
LIN {X 0,Y 551.888,Z 614.628,A -85,B 0,C 180,E1 -3322.869,E2 -3322.869} C_VEL
LIN {X 0,Y 551.867,Z 621.685,A -85,B 0,C 180,E1 -3324.154,E2 -3324.154} C_VEL
LIN {X 0,Y 551.725,Z 626.377,A -85,B 0,C 180,E1 -3325.252,E2 -3325.252} C_VEL
LIN {X 0,Y 551.75,Z 629.961,A -85,B 0,C 180,E1 -3326.349,E2 -3326.349} C_VEL
LIN {X 0,Y 551.723,Z 631.81,A -85,B 0,C 180,E1 -3327.08,E2 -3327.08} C_VEL
LIN {X 0,Y 551.645,Z 634.185,A -85,B 0,C 180,E1 -3328.541,E2 -3328.541} C_VEL
LIN {X 0,Y 551.64,Z 635,A -85,B 0,C 180,E1 -3330.001,E2 -3330.001} C_VEL
LIN {X 0,Y 551.645,Z 634.184,A -85,B 0,C 180,E1 -3331.461,E2 -3331.461} C_VEL
LIN {X 0,Y 551.724,Z 631.808,A -85,B 0,C 180,E1 -3332.922,E2 -3332.922} C_VEL
LIN {X 0,Y 551.764,Z 628.893,A -85,B 0,C 180,E1 -3334.018,E2 -3334.018} C_VEL
LIN {X 0,Y 551.724,Z 624.945,A -85,B 0,C 180,E1 -3335.117,E2 -3335.117} C_VEL
LIN {X 0,Y 551.803,Z 619.188,A -85,B 0,C 180,E1 -3336.342,E2 -3336.342} C_VEL
LIN {X 0,Y 551.927,Z 612.23,A -85,B 0,C 180,E1 -3337.5,E2 -3337.5} C_VEL
LIN {X 0,Y 552.079,Z 603.984,A -85,B 0,C 180,E1 -3338.603,E2 -3338.603} C_VEL
LIN {X 0,Y 552.222,Z 595.53,A -85,B 0,C 180,E1 -3339.524,E2 -3339.524} C_VEL
LIN {X 0,Y 552.419,Z 585.082,A -85,B 0,C 180,E1 -3340.446,E2 -3340.446} C_VEL
LIN {X 0,Y 552.557,Z 574.274,A -85,B 0,C 180,E1 -3341.215,E2 -3341.215} C_VEL
LIN {X 0,Y 552.783,Z 563.389,A -85,B 0,C 180,E1 -3341.831,E2 -3341.831} C_VEL
LIN {X 0,Y 552.909,Z 551.74,A -85,B 0,C 180,E1 -3342.34,E2 -3342.34} C_VEL
LIN {X 0,Y 553.061,Z 538.311,A -85,B 0,C 180,E1 -3342.756,E2 -3342.756} C_VEL
LIN {X 0,Y 553.196,Z 525.024,A -85,B 0,C 180,E1 -3343.01,E2 -3343.01} C_VEL
LIN {X 0,Y 553.401,Z 429.625,A -85,B 0,C 180,E1 -3344.253,E2 -3344.253} C_VEL
LIN {X 0,Y 552.381,Z 422.765,A -85,B 0,C 180,E1 -3344.393,E2 -3344.393} C_VEL
LIN {X 0,Y 552.64,Z 402.088,A -85,B 0,C 180,E1 -3347.486,E2 -3347.486} C_VEL
LIN {X 0,Y 552.959,Z 382.345,A -85,B 0,C 180,E1 -3350.459,E2 -3350.459} C_VEL
LIN {X 0,Y 553.112,Z 368.301,A -85,B 0,C 180,E1 -3352.605,E2 -3352.605} C_VEL
LIN {X 0,Y 552.128,Z 362.715,A -85,B 0,C 180,E1 -3353.537,E2 -3353.537} C_VEL
LIN {X 0,Y 552.136,Z 362.711,A -85,B 0,C 180,E1 -3355.645,E2 -3355.645} C_VEL
LIN {X 0,Y 552.13,Z 362.707,A -85,B 0,C 180,E1 -3358.563,E2 -3358.563} C_VEL
LIN {X 0,Y 552.117,Z 362.713,A -85,B 0,C 180,E1 -3361.476,E2 -3361.476} C_VEL
LIN {X 0,Y 552.142,Z 362.703,A -85,B 0,C 180,E1 -3364.171,E2 -3364.171} C_VEL
LIN {X 0,Y 552.111,Z 362.711,A -85,B 0,C 180,E1 -3366.747,E2 -3366.747} C_VEL
LIN {X 0,Y 552.139,Z 362.708,A -85,B 0,C 180,E1 -3369.527,E2 -3369.527} C_VEL
LIN {X 0,Y 552.135,Z 362.706,A -85,B 0,C 180,E1 -3372.426,E2 -3372.426} C_VEL
LIN {X 0,Y 552.104,Z 362.71,A -85,B 0,C 180,E1 -3375.563,E2 -3375.563} C_VEL
LIN {X 0,Y 552.126,Z 362.709,A -85,B 0,C 180,E1 -3378.554,E2 -3378.554} C_VEL
LIN {X 0,Y 552.121,Z 362.707,A -85,B 0,C 180,E1 -3381.411,E2 -3381.411} C_VEL
LIN {X 0,Y 552.09,Z 362.71,A -85,B 0,C 180,E1 -3384.157,E2 -3384.157} C_VEL
LIN {X 0,Y 552.121,Z 362.714,A -85,B 0,C 180,E1 -3386.814,E2 -3386.814} C_VEL
LIN {X 0,Y 552.107,Z 362.706,A -85,B 0,C 180,E1 -3389.391,E2 -3389.391} C_VEL
LIN {X 0,Y 552.108,Z 362.707,A -85,B 0,C 180,E1 -3391.902,E2 -3391.902} C_VEL
LIN {X 0,Y 552.161,Z 362.709,A -85,B 0,C 180,E1 -3394.65,E2 -3394.65} C_VEL
LIN {X 0,Y 552.098,Z 362.707,A -85,B 0,C 180,E1 -3397.549,E2 -3397.549} C_VEL
LIN {X 0,Y 552.151,Z 362.71,A -85,B 0,C 180,E1 -3400.375,E2 -3400.375} C_VEL
LIN {X 0,Y 552.161,Z 362.702,A -85,B 0,C 180,E1 -3402.977,E2 -3402.977} C_VEL
LIN {X 0,Y 552.14,Z 362.705,A -85,B 0,C 180,E1 -3406.005,E2 -3406.005} C_VEL
LIN {X 0,Y 552.168,Z 362.699,A -85,B 0,C 180,E1 -3408.994,E2 -3408.994} C_VEL
LIN {X 0,Y 552.163,Z 362.705,A -85,B 0,C 180,E1 -3411.952,E2 -3411.952} C_VEL
LIN {X 0,Y 552.233,Z 362.692,A -85,B 0,C 180,E1 -3414.889,E2 -3414.889} C_VEL
LIN {X 0,Y 552.23,Z 362.695,A -85,B 0,C 180,E1 -3417.812,E2 -3417.812} C_VEL
LIN {X 0,Y 552.247,Z 362.69,A -85,B 0,C 180,E1 -3420.729,E2 -3420.729} C_VEL
LIN {X 0,Y 552.21,Z 362.694,A -85,B 0,C 180,E1 -3422.918,E2 -3422.918} C_VEL
LIN {X 0,Y 552.205,Z 362.703,A -85,B 0,C 180,E1 -3425.844,E2 -3425.844} C_VEL
LIN {X 0,Y 552.163,Z 362.7,A -85,B 0,C 180,E1 -3428.786,E2 -3428.786} C_VEL
LIN {X 0,Y 552.169,Z 362.708,A -85,B 0,C 180,E1 -3431.75,E2 -3431.75} C_VEL
LIN {X 0,Y 552.143,Z 362.703,A -85,B 0,C 180,E1 -3434.748,E2 -3434.748} C_VEL
LIN {X 0,Y 552.115,Z 362.715,A -85,B 0,C 180,E1 -3437.789,E2 -3437.789} C_VEL
LIN {X 0,Y 552.135,Z 362.707,A -85,B 0,C 180,E1 -3440.101,E2 -3440.101} C_VEL
LIN {X 0,Y 552.099,Z 362.709,A -85,B 0,C 180,E1 -3442.451,E2 -3442.451} C_VEL
LIN {X 0,Y 552.162,Z 362.708,A -85,B 0,C 180,E1 -3445.35,E2 -3445.35} C_VEL
LIN {X 0,Y 552.111,Z 362.71,A -85,B 0,C 180,E1 -3448.098,E2 -3448.098} C_VEL
LIN {X 0,Y 552.108,Z 362.71,A -85,B 0,C 180,E1 -3450.613,E2 -3450.613} C_VEL
LIN {X 0,Y 552.15,Z 362.791,A -85,B 0,C 180,E1 -3451.913,E2 -3451.913} C_VEL
LIN {X 0,Y 552.609,Z 366.609,A -85,B 0,C 180,E1 -3452.647,E2 -3452.647} C_VEL
LIN {X 0,Y 551.912,Z 369.575,A -85,B 0,C 180,E1 -3453.172,E2 -3453.172} C_VEL
LIN {X 0,Y 546.122,Z 379.772,A -85,B 0,C 180,E1 -3454.845,E2 -3454.845} C_VEL
LIN {X 0,Y 545.387,Z 382.776,A -85,B 0,C 180,E1 -3455.377,E2 -3455.377} C_VEL
LIN {X 0,Y 545.205,Z 394.27,A -85,B 0,C 180,E1 -3457.494,E2 -3457.494} C_VEL
LIN {X 0,Y 546.568,Z 403.462,A -85,B 0,C 180,E1 -3457.66,E2 -3457.66} C_VEL
LIN {X 0,Y 546.202,Z 501.275,A -85,B 0,C 180,E1 -3458.969,E2 -3458.969} C_VEL
LIN {X 0,Y 546.057,Z 514.922,A -85,B 0,C 180,E1 -3459.308,E2 -3459.308} C_VEL
LIN {X 0,Y 545.871,Z 527.145,A -85,B 0,C 180,E1 -3459.767,E2 -3459.767} C_VEL
LIN {X 0,Y 545.669,Z 539.387,A -85,B 0,C 180,E1 -3460.386,E2 -3460.386} C_VEL
LIN {X 0,Y 545.482,Z 550.076,A -85,B 0,C 180,E1 -3461.078,E2 -3461.078} C_VEL
LIN {X 0,Y 545.235,Z 560.911,A -85,B 0,C 180,E1 -3461.959,E2 -3461.959} C_VEL
LIN {X 0,Y 545.064,Z 570.084,A -85,B 0,C 180,E1 -3462.878,E2 -3462.878} C_VEL
LIN {X 0,Y 544.901,Z 578.634,A -85,B 0,C 180,E1 -3463.926,E2 -3463.926} C_VEL
LIN {X 0,Y 544.795,Z 585.886,A -85,B 0,C 180,E1 -3465.03,E2 -3465.03} C_VEL
LIN {X 0,Y 544.709,Z 592.354,A -85,B 0,C 180,E1 -3466.264,E2 -3466.264} C_VEL
LIN {X 0,Y 544.676,Z 596.792,A -85,B 0,C 180,E1 -3467.348,E2 -3467.348} C_VEL
LIN {X 0,Y 544.651,Z 600.258,A -85,B 0,C 180,E1 -3468.454,E2 -3468.454} C_VEL
LIN {X 0,Y 544.56,Z 603.181,A -85,B 0,C 180,E1 -3469.812,E2 -3469.812} C_VEL
LIN {X 0,Y 544.541,Z 604.401,A -85,B 0,C 180,E1 -3470.771,E2 -3470.771} C_VEL
LIN {X 0,Y 544.525,Z 604.983,A -85,B 0,C 180,E1 -3471.935,E2 -3471.935} C_VEL
LIN {X 0,Y 544.56,Z 604.555,A -85,B 0,C 180,E1 -3473.146,E2 -3473.146} C_VEL
LIN {X 0,Y 544.569,Z 602.802,A -85,B 0,C 180,E1 -3474.496,E2 -3474.496} C_VEL
LIN {X 0,Y 544.622,Z 600.139,A -85,B 0,C 180,E1 -3475.678,E2 -3475.678} C_VEL
LIN {X 0,Y 544.647,Z 595.798,A -85,B 0,C 180,E1 -3477.008,E2 -3477.008} C_VEL
LIN {X 0,Y 544.749,Z 591.224,A -85,B 0,C 180,E1 -3478.064,E2 -3478.064} C_VEL
LIN {X 0,Y 544.834,Z 585.346,A -85,B 0,C 180,E1 -3479.152,E2 -3479.152} C_VEL
LIN {X 0,Y 544.949,Z 578.149,A -85,B 0,C 180,E1 -3480.229,E2 -3480.229} C_VEL
LIN {X 0,Y 545.09,Z 569.072,A -85,B 0,C 180,E1 -3481.322,E2 -3481.322} C_VEL
LIN {X 0,Y 545.269,Z 559.61,A -85,B 0,C 180,E1 -3482.249,E2 -3482.249} C_VEL
LIN {X 0,Y 545.521,Z 548.419,A -85,B 0,C 180,E1 -3483.127,E2 -3483.127} C_VEL
LIN {X 0,Y 545.697,Z 537.243,A -85,B 0,C 180,E1 -3483.825,E2 -3483.825} C_VEL
LIN {X 0,Y 545.919,Z 525.203,A -85,B 0,C 180,E1 -3484.407,E2 -3484.407} C_VEL
LIN {X 0,Y 546.068,Z 512.047,A -85,B 0,C 180,E1 -3484.866,E2 -3484.866} C_VEL
LIN {X 0,Y 546.225,Z 499.547,A -85,B 0,C 180,E1 -3485.154,E2 -3485.154} C_VEL
LIN {X 0,Y 546.396,Z 401.236,A -85,B 0,C 180,E1 -3486.464,E2 -3486.464} C_VEL
LIN {X 0,Y 545.175,Z 394.271,A -85,B 0,C 180,E1 -3486.595,E2 -3486.595} C_VEL
LIN {X 0,Y 545.466,Z 378.812,A -85,B 0,C 180,E1 -3489.445,E2 -3489.445} C_VEL
LIN {X 0,Y 545.623,Z 367.244,A -85,B 0,C 180,E1 -3491.604,E2 -3491.604} C_VEL
LIN {X 0,Y 545.137,Z 363.585,A -85,B 0,C 180,E1 -3492.322,E2 -3492.322} C_VEL
LIN {X 0,Y 545.102,Z 363.582,A -85,B 0,C 180,E1 -3495.819,E2 -3495.819} C_VEL
LIN {X 0,Y 545.124,Z 363.582,A -85,B 0,C 180,E1 -3498.849,E2 -3498.849} C_VEL
LIN {X 0,Y 545.134,Z 363.577,A -85,B 0,C 180,E1 -3501.846,E2 -3501.846} C_VEL
LIN {X 0,Y 545.206,Z 363.57,A -85,B 0,C 180,E1 -3504.822,E2 -3504.822} C_VEL
LIN {X 0,Y 545.201,Z 363.569,A -85,B 0,C 180,E1 -3507.783,E2 -3507.783} C_VEL
LIN {X 0,Y 545.217,Z 363.568,A -85,B 0,C 180,E1 -3510.738,E2 -3510.738} C_VEL
LIN {X 0,Y 545.175,Z 363.571,A -85,B 0,C 180,E1 -3512.955,E2 -3512.955} C_VEL
LIN {X 0,Y 545.173,Z 363.575,A -85,B 0,C 180,E1 -3515.918,E2 -3515.918} C_VEL
LIN {X 0,Y 545.113,Z 363.579,A -85,B 0,C 180,E1 -3518.899,E2 -3518.899} C_VEL
LIN {X 0,Y 545.138,Z 363.581,A -85,B 0,C 180,E1 -3521.903,E2 -3521.903} C_VEL
LIN {X 0,Y 545.087,Z 363.581,A -85,B 0,C 180,E1 -3524.942,E2 -3524.942} C_VEL
LIN {X 0,Y 545.082,Z 363.591,A -85,B 0,C 180,E1 -3528.025,E2 -3528.025} C_VEL
LIN {X 0,Y 545.093,Z 363.584,A -85,B 0,C 180,E1 -3530.371,E2 -3530.371} C_VEL
LIN {X 0,Y 545.081,Z 363.586,A -85,B 0,C 180,E1 -3533.558,E2 -3533.558} C_VEL
LIN {X 0,Y 545.079,Z 363.589,A -85,B 0,C 180,E1 -3535.999,E2 -3535.999} C_VEL
LIN {X 0,Y 545.09,Z 363.581,A -85,B 0,C 180,E1 -3538.747,E2 -3538.747} C_VEL
LIN {X 0,Y 545.077,Z 363.592,A -85,B 0,C 180,E1 -3541.681,E2 -3541.681} C_VEL
LIN {X 0,Y 545.08,Z 363.582,A -85,B 0,C 180,E1 -3544.562,E2 -3544.562} C_VEL
LIN {X 0,Y 545.036,Z 363.592,A -85,B 0,C 180,E1 -3547.302,E2 -3547.302} C_VEL
LIN {X 0,Y 545.072,Z 363.585,A -85,B 0,C 180,E1 -3550.14,E2 -3550.14} C_VEL
LIN {X 0,Y 545.081,Z 363.585,A -85,B 0,C 180,E1 -3553.105,E2 -3553.105} C_VEL
LIN {X 0,Y 545.061,Z 363.587,A -85,B 0,C 180,E1 -3556.223,E2 -3556.223} C_VEL
LIN {X 0,Y 545.166,Z 363.703,A -85,B 0,C 180,E1 -3557.937,E2 -3557.937} C_VEL
LIN {X 0,Y 545.541,Z 368.986,A -85,B 0,C 180,E1 -3558.927,E2 -3558.927} C_VEL
LIN {X 0,Y 545.367,Z 385.08,A -85,B 0,C 180,E1 -3561.819,E2 -3561.819} C_VEL
LIN {X 0,Y 545.201,Z 394.421,A -85,B 0,C 180,E1 -3563.507,E2 -3563.507} C_VEL
LIN {X 0,Y 546.525,Z 403.132,A -85,B 0,C 180,E1 -3563.658,E2 -3563.658} C_VEL
LIN {X 0,Y 546.189,Z 500.204,A -85,B 0,C 180,E1 -3564.956,E2 -3564.956} C_VEL
LIN {X 0,Y 546.087,Z 510.408,A -85,B 0,C 180,E1 -3565.185,E2 -3565.185} C_VEL
LIN {X 0,Y 545.973,Z 520.337,A -85,B 0,C 180,E1 -3565.501,E2 -3565.501} C_VEL
LIN {X 0,Y 545.806,Z 529.498,A -85,B 0,C 180,E1 -3565.88,E2 -3565.88} C_VEL
LIN {X 0,Y 545.656,Z 538.957,A -85,B 0,C 180,E1 -3566.369,E2 -3566.369} C_VEL
LIN {X 0,Y 545.497,Z 548.348,A -85,B 0,C 180,E1 -3566.965,E2 -3566.965} C_VEL
LIN {X 0,Y 545.333,Z 556.168,A -85,B 0,C 180,E1 -3567.558,E2 -3567.558} C_VEL
LIN {X 0,Y 545.172,Z 564.432,A -85,B 0,C 180,E1 -3568.299,E2 -3568.299} C_VEL
LIN {X 0,Y 545.077,Z 570.678,A -85,B 0,C 180,E1 -3568.953,E2 -3568.953} C_VEL
LIN {X 0,Y 544.94,Z 577.629,A -85,B 0,C 180,E1 -3569.803,E2 -3569.803} C_VEL
LIN {X 0,Y 544.797,Z 583.479,A -85,B 0,C 180,E1 -3570.645,E2 -3570.645} C_VEL
LIN {X 0,Y 544.717,Z 589.513,A -85,B 0,C 180,E1 -3571.696,E2 -3571.696} C_VEL
LIN {X 0,Y 544.676,Z 593.993,A -85,B 0,C 180,E1 -3572.649,E2 -3572.649} C_VEL
LIN {X 0,Y 544.701,Z 597.512,A -85,B 0,C 180,E1 -3573.568,E2 -3573.568} C_VEL
LIN {X 0,Y 544.621,Z 601.065,A -85,B 0,C 180,E1 -3574.796,E2 -3574.796} C_VEL
LIN {X 0,Y 544.579,Z 602.796,A -85,B 0,C 180,E1 -3575.608,E2 -3575.608} C_VEL
LIN {X 0,Y 544.583,Z 604.042,A -85,B 0,C 180,E1 -3576.418,E2 -3576.418} C_VEL
LIN {X 0,Y 544.547,Z 604.708,A -85,B 0,C 180,E1 -3577.22,E2 -3577.22} C_VEL
LIN {X 0,Y 544.56,Z 604.929,A -85,B 0,C 180,E1 -3578.31,E2 -3578.31} C_VEL
LIN {X 0,Y 544.556,Z 604.112,A -85,B 0,C 180,E1 -3579.607,E2 -3579.607} C_VEL
LIN {X 0,Y 544.572,Z 602.921,A -85,B 0,C 180,E1 -3580.404,E2 -3580.404} C_VEL
LIN {X 0,Y 544.644,Z 599.344,A -85,B 0,C 180,E1 -3581.959,E2 -3581.959} C_VEL
LIN {X 0,Y 544.667,Z 595.315,A -85,B 0,C 180,E1 -3583.122,E2 -3583.122} C_VEL
LIN {X 0,Y 544.708,Z 590.102,A -85,B 0,C 180,E1 -3584.279,E2 -3584.279} C_VEL
LIN {X 0,Y 544.777,Z 585.924,A -85,B 0,C 180,E1 -3585.048,E2 -3585.048} C_VEL
LIN {X 0,Y 544.894,Z 579.7,A -85,B 0,C 180,E1 -3586.005,E2 -3586.005} C_VEL
LIN {X 0,Y 544.971,Z 573.89,A -85,B 0,C 180,E1 -3586.767,E2 -3586.767} C_VEL
LIN {X 0,Y 545.149,Z 567.096,A -85,B 0,C 180,E1 -3587.529,E2 -3587.529} C_VEL
LIN {X 0,Y 545.293,Z 558.023,A -85,B 0,C 180,E1 -3588.378,E2 -3588.378} C_VEL
LIN {X 0,Y 545.466,Z 549.502,A -85,B 0,C 180,E1 -3589.044,E2 -3589.044} C_VEL
LIN {X 0,Y 545.622,Z 540.859,A -85,B 0,C 180,E1 -3589.611,E2 -3589.611} C_VEL
LIN {X 0,Y 545.796,Z 532.206,A -85,B 0,C 180,E1 -3590.083,E2 -3590.083} C_VEL
LIN {X 0,Y 545.964,Z 521.305,A -85,B 0,C 180,E1 -3590.553,E2 -3590.553} C_VEL
LIN {X 0,Y 546.091,Z 511.243,A -85,B 0,C 180,E1 -3590.883,E2 -3590.883} C_VEL
LIN {X 0,Y 546.206,Z 501.091,A -85,B 0,C 180,E1 -3591.118,E2 -3591.118} C_VEL
LIN {X 0,Y 546.373,Z 463.788,A -85,B 0,C 180,E1 -3591.633,E2 -3591.633} C_VEL
LIN {X 0,Y 546.473,Z 401.676,A -85,B 0,C 180,E1 -3592.453,E2 -3592.453} C_VEL
LIN {X 0,Y 545.225,Z 394.255,A -85,B 0,C 180,E1 -3592.594,E2 -3592.594} C_VEL
LIN {X 0,Y 545.354,Z 380.899,A -85,B 0,C 180,E1 -3595.01,E2 -3595.01} C_VEL
LIN {X 0,Y 545.504,Z 367.58,A -85,B 0,C 180,E1 -3597.415,E2 -3597.415} C_VEL
LIN {X 0,Y 545.158,Z 363.581,A -85,B 0,C 180,E1 -3598.153,E2 -3598.153} C_VEL
LIN {X 0,Y 545.208,Z 363.575,A -85,B 0,C 180,E1 -3600.739,E2 -3600.739} C_VEL
LIN {X 0,Y 545.169,Z 363.577,A -85,B 0,C 180,E1 -3602.956,E2 -3602.956} C_VEL
LIN {X 0,Y 545.163,Z 363.576,A -85,B 0,C 180,E1 -3605.92,E2 -3605.92} C_VEL
LIN {X 0,Y 545.119,Z 363.58,A -85,B 0,C 180,E1 -3608.9,E2 -3608.9} C_VEL
LIN {X 0,Y 545.126,Z 363.582,A -85,B 0,C 180,E1 -3611.904,E2 -3611.904} C_VEL
LIN {X 0,Y 545.076,Z 363.584,A -85,B 0,C 180,E1 -3614.944,E2 -3614.944} C_VEL
LIN {X 0,Y 545.075,Z 363.592,A -85,B 0,C 180,E1 -3618.026,E2 -3618.026} C_VEL
LIN {X 0,Y 545.09,Z 363.585,A -85,B 0,C 180,E1 -3620.372,E2 -3620.372} C_VEL
LIN {X 0,Y 545.128,Z 363.581,A -85,B 0,C 180,E1 -3623.557,E2 -3623.557} C_VEL
LIN {X 0,Y 545.092,Z 363.588,A -85,B 0,C 180,E1 -3626,E2 -3626} C_VEL
LIN {X 0,Y 545.084,Z 363.582,A -85,B 0,C 180,E1 -3628.75,E2 -3628.75} C_VEL
LIN {X 0,Y 545.07,Z 363.592,A -85,B 0,C 180,E1 -3631.683,E2 -3631.683} C_VEL
LIN {X 0,Y 545.076,Z 363.583,A -85,B 0,C 180,E1 -3634.564,E2 -3634.564} C_VEL
LIN {X 0,Y 545.032,Z 363.596,A -85,B 0,C 180,E1 -3637.304,E2 -3637.304} C_VEL
LIN {X 0,Y 545.069,Z 363.585,A -85,B 0,C 180,E1 -3640.143,E2 -3640.143} C_VEL
LIN {X 0,Y 545.081,Z 363.589,A -85,B 0,C 180,E1 -3643.107,E2 -3643.107} C_VEL
LIN {X 0,Y 545.06,Z 363.585,A -85,B 0,C 180,E1 -3646.225,E2 -3646.225} C_VEL
LIN {X 0,Y 545.092,Z 363.587,A -85,B 0,C 180,E1 -3648.888,E2 -3648.888} C_VEL
LIN {X 0,Y 545.05,Z 363.587,A -85,B 0,C 180,E1 -3651.764,E2 -3651.764} C_VEL
LIN {X 0,Y 545.063,Z 363.588,A -85,B 0,C 180,E1 -3654.535,E2 -3654.535} C_VEL
LIN {X 0,Y 545.079,Z 363.587,A -85,B 0,C 180,E1 -3657.214,E2 -3657.214} C_VEL
LIN {X 0,Y 545.099,Z 363.581,A -85,B 0,C 180,E1 -3659.814,E2 -3659.814} C_VEL
LIN {X 0,Y 545.1,Z 363.588,A -85,B 0,C 180,E1 -3662.826,E2 -3662.826} C_VEL
LIN {X 0,Y 545.052,Z 363.59,A -85,B 0,C 180,E1 -3665.632,E2 -3665.632} C_VEL
LIN {X 0,Y 545.069,Z 363.646,A -85,B 0,C 180,E1 -3666.311,E2 -3666.311} C_VEL
LIN {X 0,Y 546.224,Z 370.716,A -85,B 0,C 180,E1 -3667.471,E2 -3667.471} C_VEL
LIN {X 0,Y 545.887,Z 388.918,A -85,B 0,C 180,E1 -3670.287,E2 -3670.287} C_VEL
LIN {X 0,Y 545.58,Z 406.441,A -85,B 0,C 180,E1 -3672.96,E2 -3672.96} C_VEL
LIN {X 0,Y 545.372,Z 423.109,A -85,B 0,C 180,E1 -3675.447,E2 -3675.447} C_VEL
LIN {X 0,Y 546.56,Z 431.691,A -85,B 0,C 180,E1 -3675.593,E2 -3675.593} C_VEL
LIN {X 0,Y 546.241,Z 530.999,A -85,B 0,C 180,E1 -3676.918,E2 -3676.918} C_VEL
LIN {X 0,Y 546.075,Z 544.252,A -85,B 0,C 180,E1 -3677.245,E2 -3677.245} C_VEL
LIN {X 0,Y 545.887,Z 556.395,A -85,B 0,C 180,E1 -3677.689,E2 -3677.689} C_VEL
LIN {X 0,Y 545.675,Z 567.494,A -85,B 0,C 180,E1 -3678.232,E2 -3678.232} C_VEL
LIN {X 0,Y 545.525,Z 578.917,A -85,B 0,C 180,E1 -3678.953,E2 -3678.953} C_VEL
LIN {X 0,Y 545.285,Z 589.548,A -85,B 0,C 180,E1 -3679.793,E2 -3679.793} C_VEL
LIN {X 0,Y 545.083,Z 599.123,A -85,B 0,C 180,E1 -3680.726,E2 -3680.726} C_VEL
LIN {X 0,Y 544.977,Z 606.969,A -85,B 0,C 180,E1 -3681.659,E2 -3681.659} C_VEL
LIN {X 0,Y 544.822,Z 614.628,A -85,B 0,C 180,E1 -3682.776,E2 -3682.776} C_VEL
LIN {X 0,Y 544.776,Z 621.684,A -85,B 0,C 180,E1 -3684.077,E2 -3684.077} C_VEL
LIN {X 0,Y 544.629,Z 626.377,A -85,B 0,C 180,E1 -3685.19,E2 -3685.19} C_VEL
LIN {X 0,Y 544.669,Z 629.961,A -85,B 0,C 180,E1 -3686.302,E2 -3686.302} C_VEL
LIN {X 0,Y 544.65,Z 631.809,A -85,B 0,C 180,E1 -3687.042,E2 -3687.042} C_VEL
LIN {X 0,Y 544.546,Z 634.184,A -85,B 0,C 180,E1 -3688.522,E2 -3688.522} C_VEL
LIN {X 0,Y 544.541,Z 635,A -85,B 0,C 180,E1 -3690.001,E2 -3690.001} C_VEL
LIN {X 0,Y 544.546,Z 634.183,A -85,B 0,C 180,E1 -3691.48,E2 -3691.48} C_VEL
LIN {X 0,Y 544.651,Z 631.808,A -85,B 0,C 180,E1 -3692.96,E2 -3692.96} C_VEL
LIN {X 0,Y 544.684,Z 628.893,A -85,B 0,C 180,E1 -3694.07,E2 -3694.07} C_VEL
LIN {X 0,Y 544.654,Z 624.945,A -85,B 0,C 180,E1 -3695.183,E2 -3695.183} C_VEL
LIN {X 0,Y 544.74,Z 619.703,A -85,B 0,C 180,E1 -3696.328,E2 -3696.328} C_VEL
LIN {X 0,Y 544.837,Z 613.461,A -85,B 0,C 180,E1 -3697.412,E2 -3697.412} C_VEL
LIN {X 0,Y 545.004,Z 605.47,A -85,B 0,C 180,E1 -3698.529,E2 -3698.529} C_VEL
LIN {X 0,Y 545.153,Z 597.325,A -85,B 0,C 180,E1 -3699.462,E2 -3699.462} C_VEL
LIN {X 0,Y 545.365,Z 587.387,A -85,B 0,C 180,E1 -3700.395,E2 -3700.395} C_VEL
LIN {X 0,Y 545.571,Z 576.579,A -85,B 0,C 180,E1 -3701.209,E2 -3701.209} C_VEL
LIN {X 0,Y 545.748,Z 565.154,A -85,B 0,C 180,E1 -3701.891,E2 -3701.891} C_VEL
LIN {X 0,Y 545.945,Z 552.951,A -85,B 0,C 180,E1 -3702.453,E2 -3702.453} C_VEL
LIN {X 0,Y 546.133,Z 540.139,A -85,B 0,C 180,E1 -3702.874,E2 -3702.874} C_VEL
LIN {X 0,Y 546.256,Z 528.048,A -85,B 0,C 180,E1 -3703.131,E2 -3703.131} C_VEL
LIN {X 0,Y 546.439,Z 429.837,A -85,B 0,C 180,E1 -3704.435,E2 -3704.435} C_VEL
LIN {X 0,Y 545.375,Z 422.717,A -85,B 0,C 180,E1 -3704.581,E2 -3704.581} C_VEL
LIN {X 0,Y 545.739,Z 399.999,A -85,B 0,C 180,E1 -3708.004,E2 -3708.004} C_VEL
LIN {X 0,Y 546.038,Z 379.602,A -85,B 0,C 180,E1 -3711.125,E2 -3711.125} C_VEL
LIN {X 0,Y 546.132,Z 369.405,A -85,B 0,C 180,E1 -3712.71,E2 -3712.71} C_VEL
LIN {X 0,Y 545.072,Z 363.592,A -85,B 0,C 180,E1 -3713.691,E2 -3713.691} C_VEL
LIN {X 0,Y 545.086,Z 363.585,A -85,B 0,C 180,E1 -3716.001,E2 -3716.001} C_VEL
LIN {X 0,Y 545.095,Z 363.585,A -85,B 0,C 180,E1 -3718.749,E2 -3718.749} C_VEL
LIN {X 0,Y 545.064,Z 363.589,A -85,B 0,C 180,E1 -3721.679,E2 -3721.679} C_VEL
LIN {X 0,Y 545.082,Z 363.584,A -85,B 0,C 180,E1 -3724.564,E2 -3724.564} C_VEL
LIN {X 0,Y 545.043,Z 363.596,A -85,B 0,C 180,E1 -3727.304,E2 -3727.304} C_VEL
LIN {X 0,Y 545.074,Z 363.585,A -85,B 0,C 180,E1 -3730.143,E2 -3730.143} C_VEL
LIN {X 0,Y 545.084,Z 363.592,A -85,B 0,C 180,E1 -3733.107,E2 -3733.107} C_VEL
LIN {X 0,Y 545.073,Z 363.585,A -85,B 0,C 180,E1 -3736.225,E2 -3736.225} C_VEL
LIN {X 0,Y 545.087,Z 363.591,A -85,B 0,C 180,E1 -3738.886,E2 -3738.886} C_VEL
LIN {X 0,Y 545.084,Z 363.59,A -85,B 0,C 180,E1 -3740.818,E2 -3740.818} C_VEL
LIN {X 0,Y 545.047,Z 363.587,A -85,B 0,C 180,E1 -3743.62,E2 -3743.62} C_VEL
LIN {X 0,Y 545.071,Z 363.586,A -85,B 0,C 180,E1 -3746.328,E2 -3746.328} C_VEL
LIN {X 0,Y 545.071,Z 363.587,A -85,B 0,C 180,E1 -3748.952,E2 -3748.952} C_VEL
LIN {X 0,Y 545.106,Z 363.579,A -85,B 0,C 180,E1 -3751.508,E2 -3751.508} C_VEL
LIN {X 0,Y 545.099,Z 363.586,A -85,B 0,C 180,E1 -3754.492,E2 -3754.492} C_VEL
LIN {X 0,Y 545.043,Z 363.586,A -85,B 0,C 180,E1 -3757.242,E2 -3757.242} C_VEL
LIN {X 0,Y 545.123,Z 363.586,A -85,B 0,C 180,E1 -3760.415,E2 -3760.415} C_VEL
LIN {X 0,Y 545.077,Z 363.583,A -85,B 0,C 180,E1 -3763.521,E2 -3763.521} C_VEL
LIN {X 0,Y 545.1,Z 363.58,A -85,B 0,C 180,E1 -3765.82,E2 -3765.82} C_VEL
LIN {X 0,Y 545.123,Z 363.577,A -85,B 0,C 180,E1 -3768.849,E2 -3768.849} C_VEL
LIN {X 0,Y 545.134,Z 363.58,A -85,B 0,C 180,E1 -3771.847,E2 -3771.847} C_VEL
LIN {X 0,Y 545.209,Z 363.568,A -85,B 0,C 180,E1 -3774.823,E2 -3774.823} C_VEL
LIN {X 0,Y 545.202,Z 363.57,A -85,B 0,C 180,E1 -3777.784,E2 -3777.784} C_VEL
LIN {X 0,Y 545.217,Z 363.566,A -85,B 0,C 180,E1 -3780.739,E2 -3780.739} C_VEL
LIN {X 0,Y 545.177,Z 363.57,A -85,B 0,C 180,E1 -3782.956,E2 -3782.956} C_VEL
LIN {X 0,Y 545.177,Z 363.58,A -85,B 0,C 180,E1 -3785.92,E2 -3785.92} C_VEL
LIN {X 0,Y 545.122,Z 363.577,A -85,B 0,C 180,E1 -3788.9,E2 -3788.9} C_VEL
LIN {X 0,Y 545.141,Z 363.583,A -85,B 0,C 180,E1 -3791.904,E2 -3791.904} C_VEL
LIN {X 0,Y 545.092,Z 363.582,A -85,B 0,C 180,E1 -3794.944,E2 -3794.944} C_VEL
LIN {X 0,Y 545.082,Z 363.588,A -85,B 0,C 180,E1 -3798.026,E2 -3798.026} C_VEL
LIN {X 0,Y 545.1,Z 363.581,A -85,B 0,C 180,E1 -3800.372,E2 -3800.372} C_VEL
LIN {X 0,Y 545.087,Z 363.59,A -85,B 0,C 180,E1 -3803.559,E2 -3803.559} C_VEL
LIN {X 0,Y 545.086,Z 363.586,A -85,B 0,C 180,E1 -3806,E2 -3806} C_VEL
LIN {X 0,Y 545.095,Z 363.583,A -85,B 0,C 180,E1 -3808.748,E2 -3808.748} C_VEL
LIN {X 0,Y 545.093,Z 363.621,A -85,B 0,C 180,E1 -3811.763,E2 -3811.763} C_VEL
LIN {X 0,Y 545.64,Z 368.703,A -85,B 0,C 180,E1 -3812.75,E2 -3812.75} C_VEL
LIN {X 0,Y 545.387,Z 382.776,A -85,B 0,C 180,E1 -3815.377,E2 -3815.377} C_VEL
LIN {X 0,Y 544.665,Z 384.808,A -85,B 0,C 180,E1 -3815.728,E2 -3815.728} C_VEL
LIN {X 0,Y 538.926,Z 391.638,A -85,B 0,C 180,E1 -3816.8,E2 -3816.8} C_VEL
LIN {X 0,Y 538.231,Z 393.683,A -85,B 0,C 180,E1 -3817.157,E2 -3817.157} C_VEL
LIN {X 0,Y 538.214,Z 394.649,A -85,B 0,C 180,E1 -3817.311,E2 -3817.311} C_VEL
LIN {X 0,Y 539.697,Z 403.445,A -85,B 0,C 180,E1 -3817.472,E2 -3817.472} C_VEL
LIN {X 0,Y 539.307,Z 501.105,A -85,B 0,C 180,E1 -3818.795,E2 -3818.795} C_VEL
LIN {X 0,Y 539.157,Z 514.36,A -85,B 0,C 180,E1 -3819.123,E2 -3819.123} C_VEL
LIN {X 0,Y 538.956,Z 525.931,A -85,B 0,C 180,E1 -3819.547,E2 -3819.547} C_VEL
LIN {X 0,Y 538.743,Z 538.205,A -85,B 0,C 180,E1 -3820.16,E2 -3820.16} C_VEL
LIN {X 0,Y 538.528,Z 549.124,A -85,B 0,C 180,E1 -3820.861,E2 -3820.861} C_VEL
LIN {X 0,Y 538.219,Z 560.214,A -85,B 0,C 180,E1 -3821.756,E2 -3821.756} C_VEL
LIN {X 0,Y 538.018,Z 570.385,A -85,B 0,C 180,E1 -3822.786,E2 -3822.786} C_VEL
LIN {X 0,Y 537.833,Z 578.743,A -85,B 0,C 180,E1 -3823.834,E2 -3823.834} C_VEL
LIN {X 0,Y 537.693,Z 586.843,A -85,B 0,C 180,E1 -3825.104,E2 -3825.104} C_VEL
LIN {X 0,Y 537.638,Z 593.257,A -85,B 0,C 180,E1 -3826.39,E2 -3826.39} C_VEL
LIN {X 0,Y 537.572,Z 598.112,A -85,B 0,C 180,E1 -3827.678,E2 -3827.678} C_VEL
LIN {X 0,Y 537.485,Z 602.067,A -85,B 0,C 180,E1 -3829.172,E2 -3829.172} C_VEL
LIN {X 0,Y 537.44,Z 604.128,A -85,B 0,C 180,E1 -3830.492,E2 -3830.492} C_VEL
LIN {X 0,Y 537.428,Z 604.932,A -85,B 0,C 180,E1 -3831.687,E2 -3831.687} C_VEL
LIN {X 0,Y 537.449,Z 604.642,A -85,B 0,C 180,E1 -3833.02,E2 -3833.02} C_VEL
LIN {X 0,Y 537.451,Z 603.381,A -85,B 0,C 180,E1 -3834.169,E2 -3834.169} C_VEL
LIN {X 0,Y 537.515,Z 600.833,A -85,B 0,C 180,E1 -3835.46,E2 -3835.46} C_VEL
LIN {X 0,Y 537.573,Z 596.827,A -85,B 0,C 180,E1 -3836.795,E2 -3836.795} C_VEL
LIN {X 0,Y 537.663,Z 591.086,A -85,B 0,C 180,E1 -3838.173,E2 -3838.173} C_VEL
LIN {X 0,Y 537.765,Z 584.697,A -85,B 0,C 180,E1 -3839.356,E2 -3839.356} C_VEL
LIN {X 0,Y 537.893,Z 577.331,A -85,B 0,C 180,E1 -3840.446,E2 -3840.446} C_VEL
LIN {X 0,Y 538.093,Z 568.35,A -85,B 0,C 180,E1 -3841.527,E2 -3841.527} C_VEL
LIN {X 0,Y 538.298,Z 558.517,A -85,B 0,C 180,E1 -3842.485,E2 -3842.485} C_VEL
LIN {X 0,Y 538.539,Z 547.468,A -85,B 0,C 180,E1 -3843.345,E2 -3843.345} C_VEL
LIN {X 0,Y 538.782,Z 536.552,A -85,B 0,C 180,E1 -3844.024,E2 -3844.024} C_VEL
LIN {X 0,Y 539.004,Z 524.093,A -85,B 0,C 180,E1 -3844.617,E2 -3844.617} C_VEL
LIN {X 0,Y 539.201,Z 511.03,A -85,B 0,C 180,E1 -3845.065,E2 -3845.065} C_VEL
LIN {X 0,Y 539.316,Z 497.758,A -85,B 0,C 180,E1 -3845.354,E2 -3845.354} C_VEL
LIN {X 0,Y 539.528,Z 402.064,A -85,B 0,C 180,E1 -3846.641,E2 -3846.641} C_VEL
LIN {X 0,Y 538.174,Z 394.478,A -85,B 0,C 180,E1 -3846.782,E2 -3846.782} C_VEL
LIN {X 0,Y 538.506,Z 378.694,A -85,B 0,C 180,E1 -3849.732,E2 -3849.732} C_VEL
LIN {X 0,Y 538.619,Z 367.987,A -85,B 0,C 180,E1 -3851.75,E2 -3851.75} C_VEL
LIN {X 0,Y 538.098,Z 364.462,A -85,B 0,C 180,E1 -3852.448,E2 -3852.448} C_VEL
LIN {X 0,Y 538.071,Z 364.457,A -85,B 0,C 180,E1 -3855.63,E2 -3855.63} C_VEL
LIN {X 0,Y 538.084,Z 364.462,A -85,B 0,C 180,E1 -3858.701,E2 -3858.701} C_VEL
LIN {X 0,Y 538.091,Z 364.453,A -85,B 0,C 180,E1 -3861.739,E2 -3861.739} C_VEL
LIN {X 0,Y 538.163,Z 364.448,A -85,B 0,C 180,E1 -3864.754,E2 -3864.754} C_VEL
LIN {X 0,Y 538.173,Z 364.444,A -85,B 0,C 180,E1 -3867.754,E2 -3867.754} C_VEL
LIN {X 0,Y 538.187,Z 364.444,A -85,B 0,C 180,E1 -3870.747,E2 -3870.747} C_VEL
LIN {X 0,Y 538.142,Z 364.447,A -85,B 0,C 180,E1 -3872.993,E2 -3872.993} C_VEL
LIN {X 0,Y 538.126,Z 364.454,A -85,B 0,C 180,E1 -3875.996,E2 -3875.996} C_VEL
LIN {X 0,Y 538.064,Z 364.456,A -85,B 0,C 180,E1 -3879.017,E2 -3879.017} C_VEL
LIN {X 0,Y 538.086,Z 364.462,A -85,B 0,C 180,E1 -3882.061,E2 -3882.061} C_VEL
LIN {X 0,Y 538.047,Z 364.458,A -85,B 0,C 180,E1 -3885.143,E2 -3885.143} C_VEL
LIN {X 0,Y 538.033,Z 364.465,A -85,B 0,C 180,E1 -3888.269,E2 -3888.269} C_VEL
LIN {X 0,Y 538.038,Z 364.46,A -85,B 0,C 180,E1 -3890.65,E2 -3890.65} C_VEL
LIN {X 0,Y 538.005,Z 364.473,A -85,B 0,C 180,E1 -3893.887,E2 -3893.887} C_VEL
LIN {X 0,Y 538.041,Z 364.461,A -85,B 0,C 180,E1 -3896.365,E2 -3896.365} C_VEL
LIN {X 0,Y 538.036,Z 364.46,A -85,B 0,C 180,E1 -3898.934,E2 -3898.934} C_VEL
LIN {X 0,Y 538.026,Z 364.468,A -85,B 0,C 180,E1 -3901.889,E2 -3901.889} C_VEL
LIN {X 0,Y 538.03,Z 364.46,A -85,B 0,C 180,E1 -3904.62,E2 -3904.62} C_VEL
LIN {X 0,Y 538.005,Z 364.466,A -85,B 0,C 180,E1 -3907.169,E2 -3907.169} C_VEL
LIN {X 0,Y 538.045,Z 364.464,A -85,B 0,C 180,E1 -3909.793,E2 -3909.793} C_VEL
LIN {X 0,Y 538.028,Z 364.463,A -85,B 0,C 180,E1 -3912.987,E2 -3912.987} C_VEL
LIN {X 0,Y 538.024,Z 364.466,A -85,B 0,C 180,E1 -3915.924,E2 -3915.924} C_VEL
LIN {X 0,Y 538.103,Z 364.618,A -85,B 0,C 180,E1 -3917.861,E2 -3917.861} C_VEL
LIN {X 0,Y 538.549,Z 369.423,A -85,B 0,C 180,E1 -3918.772,E2 -3918.772} C_VEL
LIN {X 0,Y 538.348,Z 386.473,A -85,B 0,C 180,E1 -3921.853,E2 -3921.853} C_VEL
LIN {X 0,Y 538.185,Z 394.399,A -85,B 0,C 180,E1 -3923.313,E2 -3923.313} C_VEL
LIN {X 0,Y 539.651,Z 404.043,A -85,B 0,C 180,E1 -3923.489,E2 -3923.489} C_VEL
LIN {X 0,Y 539.281,Z 500.466,A -85,B 0,C 180,E1 -3924.797,E2 -3924.797} C_VEL
LIN {X 0,Y 539.161,Z 511.18,A -85,B 0,C 180,E1 -3925.043,E2 -3925.043} C_VEL
LIN {X 0,Y 539.005,Z 522.55,A -85,B 0,C 180,E1 -3925.423,E2 -3925.423} C_VEL
LIN {X 0,Y 538.776,Z 535.149,A -85,B 0,C 180,E1 -3925.996,E2 -3925.996} C_VEL
LIN {X 0,Y 538.586,Z 545.628,A -85,B 0,C 180,E1 -3926.627,E2 -3926.627} C_VEL
LIN {X 0,Y 538.348,Z 554.839,A -85,B 0,C 180,E1 -3927.307,E2 -3927.307} C_VEL
LIN {X 0,Y 538.175,Z 563.554,A -85,B 0,C 180,E1 -3928.082,E2 -3928.082} C_VEL
LIN {X 0,Y 538.009,Z 571.574,A -85,B 0,C 180,E1 -3928.936,E2 -3928.936} C_VEL
LIN {X 0,Y 537.897,Z 576.782,A -85,B 0,C 180,E1 -3929.577,E2 -3929.577} C_VEL
LIN {X 0,Y 537.75,Z 582.801,A -85,B 0,C 180,E1 -3930.438,E2 -3930.438} C_VEL
LIN {X 0,Y 537.651,Z 589.058,A -85,B 0,C 180,E1 -3931.523,E2 -3931.523} C_VEL
LIN {X 0,Y 537.596,Z 594.774,A -85,B 0,C 180,E1 -3932.77,E2 -3932.77} C_VEL
LIN {X 0,Y 537.612,Z 597.832,A -85,B 0,C 180,E1 -3933.61,E2 -3933.61} C_VEL
LIN {X 0,Y 537.563,Z 600.32,A -85,B 0,C 180,E1 -3934.441,E2 -3934.441} C_VEL
LIN {X 0,Y 537.486,Z 602.261,A -85,B 0,C 180,E1 -3935.265,E2 -3935.265} C_VEL
LIN {X 0,Y 537.477,Z 603.839,A -85,B 0,C 180,E1 -3936.247,E2 -3936.247} C_VEL
LIN {X 0,Y 537.448,Z 604.919,A -85,B 0,C 180,E1 -3937.714,E2 -3937.714} C_VEL
LIN {X 0,Y 537.461,Z 604.913,A -85,B 0,C 180,E1 -3938.522,E2 -3938.522} C_VEL
LIN {X 0,Y 537.459,Z 604.355,A -85,B 0,C 180,E1 -3939.325,E2 -3939.325} C_VEL
LIN {X 0,Y 537.48,Z 603.134,A -85,B 0,C 180,E1 -3940.294,E2 -3940.294} C_VEL
LIN {X 0,Y 537.489,Z 602.048,A -85,B 0,C 180,E1 -3940.92,E2 -3940.92} C_VEL
LIN {X 0,Y 537.569,Z 599.027,A -85,B 0,C 180,E1 -3942.107,E2 -3942.107} C_VEL
LIN {X 0,Y 537.584,Z 594.917,A -85,B 0,C 180,E1 -3943.285,E2 -3943.285} C_VEL
LIN {X 0,Y 537.651,Z 589.614,A -85,B 0,C 180,E1 -3944.456,E2 -3944.456} C_VEL
LIN {X 0,Y 537.775,Z 584.559,A -85,B 0,C 180,E1 -3945.363,E2 -3945.363} C_VEL
LIN {X 0,Y 537.858,Z 579.013,A -85,B 0,C 180,E1 -3946.204,E2 -3946.204} C_VEL
LIN {X 0,Y 537.95,Z 573.097,A -85,B 0,C 180,E1 -3946.976,E2 -3946.976} C_VEL
LIN {X 0,Y 538.125,Z 566.18,A -85,B 0,C 180,E1 -3947.747,E2 -3947.747} C_VEL
LIN {X 0,Y 538.261,Z 558.75,A -85,B 0,C 180,E1 -3948.455,E2 -3948.455} C_VEL
LIN {X 0,Y 538.469,Z 549.559,A -85,B 0,C 180,E1 -3949.186,E2 -3949.186} C_VEL
LIN {X 0,Y 538.672,Z 540.881,A -85,B 0,C 180,E1 -3949.76,E2 -3949.76} C_VEL
LIN {X 0,Y 538.849,Z 530.219,A -85,B 0,C 180,E1 -3950.333,E2 -3950.333} C_VEL
LIN {X 0,Y 539.045,Z 519.962,A -85,B 0,C 180,E1 -3950.762,E2 -3950.762} C_VEL
LIN {X 0,Y 539.169,Z 509.36,A -85,B 0,C 180,E1 -3951.095,E2 -3951.095} C_VEL
LIN {X 0,Y 539.296,Z 498.1,A -85,B 0,C 180,E1 -3951.334,E2 -3951.334} C_VEL
LIN {X 0,Y 539.601,Z 402.562,A -85,B 0,C 180,E1 -3952.622,E2 -3952.622} C_VEL
LIN {X 0,Y 538.225,Z 394.385,A -85,B 0,C 180,E1 -3952.789,E2 -3952.789} C_VEL
LIN {X 0,Y 538.349,Z 381.481,A -85,B 0,C 180,E1 -3955.132,E2 -3955.132} C_VEL
LIN {X 0,Y 538.501,Z 369.013,A -85,B 0,C 180,E1 -3957.382,E2 -3957.382} C_VEL
LIN {X 0,Y 538.115,Z 364.458,A -85,B 0,C 180,E1 -3958.222,E2 -3958.222} C_VEL
LIN {X 0,Y 538.177,Z 364.451,A -85,B 0,C 180,E1 -3960.748,E2 -3960.748} C_VEL
LIN {X 0,Y 538.135,Z 364.453,A -85,B 0,C 180,E1 -3962.994,E2 -3962.994} C_VEL
LIN {X 0,Y 538.116,Z 364.455,A -85,B 0,C 180,E1 -3965.997,E2 -3965.997} C_VEL
LIN {X 0,Y 538.068,Z 364.458,A -85,B 0,C 180,E1 -3969.018,E2 -3969.018} C_VEL
LIN {X 0,Y 538.074,Z 364.463,A -85,B 0,C 180,E1 -3972.063,E2 -3972.063} C_VEL
LIN {X 0,Y 538.037,Z 364.461,A -85,B 0,C 180,E1 -3975.144,E2 -3975.144} C_VEL
LIN {X 0,Y 538.026,Z 364.468,A -85,B 0,C 180,E1 -3978.27,E2 -3978.27} C_VEL
LIN {X 0,Y 538.033,Z 364.462,A -85,B 0,C 180,E1 -3980.652,E2 -3980.652} C_VEL
LIN {X 0,Y 538.044,Z 364.459,A -85,B 0,C 180,E1 -3983.071,E2 -3983.071} C_VEL
LIN {X 0,Y 538.054,Z 364.465,A -85,B 0,C 180,E1 -3985.678,E2 -3985.678} C_VEL
LIN {X 0,Y 538.04,Z 364.465,A -85,B 0,C 180,E1 -3988.05,E2 -3988.05} C_VEL
LIN {X 0,Y 538.02,Z 364.463,A -85,B 0,C 180,E1 -3990.627,E2 -3990.627} C_VEL
LIN {X 0,Y 538.036,Z 364.465,A -85,B 0,C 180,E1 -3993.284,E2 -3993.284} C_VEL
LIN {X 0,Y 538.02,Z 364.465,A -85,B 0,C 180,E1 -3996.003,E2 -3996.003} C_VEL
LIN {X 0,Y 538.011,Z 364.465,A -85,B 0,C 180,E1 -3998.831,E2 -3998.831} C_VEL
LIN {X 0,Y 538.031,Z 364.463,A -85,B 0,C 180,E1 -4001.881,E2 -4001.881} C_VEL
LIN {X 0,Y 538.025,Z 364.469,A -85,B 0,C 180,E1 -4005.142,E2 -4005.142} C_VEL
LIN {X 0,Y 538.035,Z 364.461,A -85,B 0,C 180,E1 -4008.229,E2 -4008.229} C_VEL
LIN {X 0,Y 538.011,Z 364.471,A -85,B 0,C 180,E1 -4011.171,E2 -4011.171} C_VEL
LIN {X 0,Y 538.026,Z 364.462,A -85,B 0,C 180,E1 -4014.084,E2 -4014.084} C_VEL
LIN {X 0,Y 538.028,Z 364.469,A -85,B 0,C 180,E1 -4016.729,E2 -4016.729} C_VEL
LIN {X 0,Y 538.035,Z 364.462,A -85,B 0,C 180,E1 -4019.555,E2 -4019.555} C_VEL
LIN {X 0,Y 538.046,Z 364.46,A -85,B 0,C 180,E1 -4021.952,E2 -4021.952} C_VEL
LIN {X 0,Y 538.075,Z 364.463,A -85,B 0,C 180,E1 -4024.469,E2 -4024.469} C_VEL
LIN {X 0,Y 538.042,Z 364.587,A -85,B 0,C 180,E1 -4026.157,E2 -4026.157} C_VEL
LIN {X 0,Y 539.302,Z 372.229,A -85,B 0,C 180,E1 -4027.433,E2 -4027.433} C_VEL
LIN {X 0,Y 538.927,Z 389.777,A -85,B 0,C 180,E1 -4030.182,E2 -4030.182} C_VEL
LIN {X 0,Y 538.576,Z 407.549,A -85,B 0,C 180,E1 -4032.927,E2 -4032.927} C_VEL
LIN {X 0,Y 538.348,Z 422.672,A -85,B 0,C 180,E1 -4035.24,E2 -4035.24} C_VEL
LIN {X 0,Y 539.701,Z 432.631,A -85,B 0,C 180,E1 -4035.423,E2 -4035.423} C_VEL
LIN {X 0,Y 539.318,Z 530.751,A -85,B 0,C 180,E1 -4036.747,E2 -4036.747} C_VEL
LIN {X 0,Y 539.144,Z 544.063,A -85,B 0,C 180,E1 -4037.078,E2 -4037.078} C_VEL
LIN {X 0,Y 538.939,Z 556.252,A -85,B 0,C 180,E1 -4037.528,E2 -4037.528} C_VEL
LIN {X 0,Y 538.72,Z 567.415,A -85,B 0,C 180,E1 -4038.079,E2 -4038.079} C_VEL
LIN {X 0,Y 538.526,Z 578.863,A -85,B 0,C 180,E1 -4038.807,E2 -4038.807} C_VEL
LIN {X 0,Y 538.271,Z 589.538,A -85,B 0,C 180,E1 -4039.659,E2 -4039.659} C_VEL
LIN {X 0,Y 538.066,Z 599.123,A -85,B 0,C 180,E1 -4040.604,E2 -4040.604} C_VEL
LIN {X 0,Y 537.92,Z 606.969,A -85,B 0,C 180,E1 -4041.549,E2 -4041.549} C_VEL
LIN {X 0,Y 537.753,Z 614.627,A -85,B 0,C 180,E1 -4042.68,E2 -4042.68} C_VEL
LIN {X 0,Y 537.693,Z 621.684,A -85,B 0,C 180,E1 -4043.999,E2 -4043.999} C_VEL
LIN {X 0,Y 537.54,Z 626.377,A -85,B 0,C 180,E1 -4045.126,E2 -4045.126} C_VEL
LIN {X 0,Y 537.591,Z 629.961,A -85,B 0,C 180,E1 -4046.253,E2 -4046.253} C_VEL
LIN {X 0,Y 537.551,Z 631.809,A -85,B 0,C 180,E1 -4047.003,E2 -4047.003} C_VEL
LIN {X 0,Y 537.451,Z 634.183,A -85,B 0,C 180,E1 -4048.502,E2 -4048.502} C_VEL
LIN {X 0,Y 537.442,Z 635,A -85,B 0,C 180,E1 -4050.001,E2 -4050.001} C_VEL
LIN {X 0,Y 537.451,Z 634.182,A -85,B 0,C 180,E1 -4051.5,E2 -4051.5} C_VEL
LIN {X 0,Y 537.551,Z 631.808,A -85,B 0,C 180,E1 -4052.999,E2 -4052.999} C_VEL
LIN {X 0,Y 537.603,Z 628.892,A -85,B 0,C 180,E1 -4054.124,E2 -4054.124} C_VEL
LIN {X 0,Y 537.588,Z 624.944,A -85,B 0,C 180,E1 -4055.252,E2 -4055.252} C_VEL
LIN {X 0,Y 537.651,Z 620.08,A -85,B 0,C 180,E1 -4056.336,E2 -4056.336} C_VEL
LIN {X 0,Y 537.792,Z 613.46,A -85,B 0,C 180,E1 -4057.51,E2 -4057.51} C_VEL
LIN {X 0,Y 537.97,Z 605.47,A -85,B 0,C 180,E1 -4058.641,E2 -4058.641} C_VEL
LIN {X 0,Y 538.143,Z 597.324,A -85,B 0,C 180,E1 -4059.586,E2 -4059.586} C_VEL
LIN {X 0,Y 538.362,Z 587.368,A -85,B 0,C 180,E1 -4060.532,E2 -4060.532} C_VEL
LIN {X 0,Y 538.556,Z 577.516,A -85,B 0,C 180,E1 -4061.289,E2 -4061.289} C_VEL
LIN {X 0,Y 538.734,Z 566.414,A -85,B 0,C 180,E1 -4061.974,E2 -4061.974} C_VEL
LIN {X 0,Y 538.973,Z 553.916,A -85,B 0,C 180,E1 -4062.569,E2 -4062.569} C_VEL
LIN {X 0,Y 539.197,Z 540.822,A -85,B 0,C 180,E1 -4063.018,E2 -4063.018} C_VEL
LIN {X 0,Y 539.36,Z 527.729,A -85,B 0,C 180,E1 -4063.302,E2 -4063.302} C_VEL
LIN {X 0,Y 539.559,Z 430.531,A -85,B 0,C 180,E1 -4064.608,E2 -4064.608} C_VEL
LIN {X 0,Y 538.345,Z 422.631,A -85,B 0,C 180,E1 -4064.759,E2 -4064.759} C_VEL
LIN {X 0,Y 538.745,Z 400.844,A -85,B 0,C 180,E1 -4068.086,E2 -4068.086} C_VEL
LIN {X 0,Y 539.081,Z 380.687,A -85,B 0,C 180,E1 -4071.21,E2 -4071.21} C_VEL
LIN {X 0,Y 539.163,Z 370.51,A -85,B 0,C 180,E1 -4072.818,E2 -4072.818} C_VEL
LIN {X 0,Y 538.043,Z 364.467,A -85,B 0,C 180,E1 -4073.844,E2 -4073.844} C_VEL
LIN {X 0,Y 538.048,Z 364.46,A -85,B 0,C 180,E1 -4076.367,E2 -4076.367} C_VEL
LIN {X 0,Y 538.037,Z 364.467,A -85,B 0,C 180,E1 -4078.934,E2 -4078.934} C_VEL
LIN {X 0,Y 538.017,Z 364.465,A -85,B 0,C 180,E1 -4081.888,E2 -4081.888} C_VEL
LIN {X 0,Y 538.031,Z 364.463,A -85,B 0,C 180,E1 -4084.62,E2 -4084.62} C_VEL
LIN {X 0,Y 538.011,Z 364.473,A -85,B 0,C 180,E1 -4087.17,E2 -4087.17} C_VEL
LIN {X 0,Y 538.032,Z 364.463,A -85,B 0,C 180,E1 -4089.797,E2 -4089.797} C_VEL
LIN {X 0,Y 538.024,Z 364.468,A -85,B 0,C 180,E1 -4092.786,E2 -4092.786} C_VEL
LIN {X 0,Y 538.038,Z 364.468,A -85,B 0,C 180,E1 -4095.141,E2 -4095.141} C_VEL
LIN {X 0,Y 538.036,Z 364.461,A -85,B 0,C 180,E1 -4098.227,E2 -4098.227} C_VEL
LIN {X 0,Y 538.017,Z 364.467,A -85,B 0,C 180,E1 -4101.17,E2 -4101.17} C_VEL
LIN {X 0,Y 537.999,Z 364.465,A -85,B 0,C 180,E1 -4104.089,E2 -4104.089} C_VEL
LIN {X 0,Y 538.036,Z 364.467,A -85,B 0,C 180,E1 -4106.728,E2 -4106.728} C_VEL
LIN {X 0,Y 538.032,Z 364.458,A -85,B 0,C 180,E1 -4109.556,E2 -4109.556} C_VEL
LIN {X 0,Y 538.042,Z 364.46,A -85,B 0,C 180,E1 -4111.95,E2 -4111.95} C_VEL
LIN {X 0,Y 538.075,Z 364.461,A -85,B 0,C 180,E1 -4114.467,E2 -4114.467} C_VEL
LIN {X 0,Y 537.999,Z 364.463,A -85,B 0,C 180,E1 -4117.739,E2 -4117.739} C_VEL
LIN {X 0,Y 538.085,Z 364.458,A -85,B 0,C 180,E1 -4120.148,E2 -4120.148} C_VEL
LIN {X 0,Y 538.029,Z 364.461,A -85,B 0,C 180,E1 -4123.299,E2 -4123.299} C_VEL
LIN {X 0,Y 538.069,Z 364.454,A -85,B 0,C 180,E1 -4125.631,E2 -4125.631} C_VEL
LIN {X 0,Y 538.083,Z 364.456,A -85,B 0,C 180,E1 -4128.702,E2 -4128.702} C_VEL
LIN {X 0,Y 538.091,Z 364.456,A -85,B 0,C 180,E1 -4131.74,E2 -4131.74} C_VEL
LIN {X 0,Y 538.167,Z 364.446,A -85,B 0,C 180,E1 -4134.755,E2 -4134.755} C_VEL
LIN {X 0,Y 538.173,Z 364.445,A -85,B 0,C 180,E1 -4137.755,E2 -4137.755} C_VEL
LIN {X 0,Y 538.187,Z 364.441,A -85,B 0,C 180,E1 -4140.748,E2 -4140.748} C_VEL
LIN {X 0,Y 538.144,Z 364.446,A -85,B 0,C 180,E1 -4142.995,E2 -4142.995} C_VEL
LIN {X 0,Y 538.13,Z 364.456,A -85,B 0,C 180,E1 -4145.997,E2 -4145.997} C_VEL
LIN {X 0,Y 538.073,Z 364.456,A -85,B 0,C 180,E1 -4149.018,E2 -4149.018} C_VEL
LIN {X 0,Y 538.089,Z 364.459,A -85,B 0,C 180,E1 -4152.062,E2 -4152.062} C_VEL
LIN {X 0,Y 538.052,Z 364.46,A -85,B 0,C 180,E1 -4155.144,E2 -4155.144} C_VEL
LIN {X 0,Y 538.035,Z 364.463,A -85,B 0,C 180,E1 -4158.27,E2 -4158.27} C_VEL
LIN {X 0,Y 538.045,Z 364.46,A -85,B 0,C 180,E1 -4160.651,E2 -4160.651} C_VEL
LIN {X 0,Y 538.01,Z 364.469,A -85,B 0,C 180,E1 -4163.888,E2 -4163.888} C_VEL
LIN {X 0,Y 538.047,Z 364.461,A -85,B 0,C 180,E1 -4166.367,E2 -4166.367} C_VEL
LIN {X 0,Y 538.036,Z 364.464,A -85,B 0,C 180,E1 -4168.933,E2 -4168.933} C_VEL
LIN {X 0,Y 538.055,Z 364.511,A -85,B 0,C 180,E1 -4171.625,E2 -4171.625} C_VEL
LIN {X 0,Y 538.707,Z 369.232,A -85,B 0,C 180,E1 -4172.558,E2 -4172.558} C_VEL
LIN {X 0,Y 538.376,Z 386.032,A -85,B 0,C 180,E1 -4175.732,E2 -4175.732} C_VEL
LIN {X 0,Y 538.231,Z 393.683,A -85,B 0,C 180,E1 -4177.157,E2 -4177.157} C_VEL
LIN {X 0,Y 537.794,Z 395.191,A -85,B 0,C 180,E1 -4177.281,E2 -4177.281} C_VEL
LIN {X 0,Y 535.78,Z 399.602,A -85,B 0,C 180,E1 -4177.31,E2 -4177.31} C_VEL
LIN {X 0,Y 533.199,Z 407.769,A -85,B 0,C 180,E1 -4177.341,E2 -4177.341} C_VEL
LIN {X 0,Y 532.543,Z 413.744,A -85,B 0,C 180,E1 -4177.377,E2 -4177.377} C_VEL
LIN {X 0,Y 532.733,Z 424.698,A -85,B 0,C 180,E1 -4177.566,E2 -4177.566} C_VEL
LIN {X 0,Y 532.403,Z 501.333,A -85,B 0,C 180,E1 -4178.624,E2 -4178.624} C_VEL
LIN {X 0,Y 532.246,Z 514.32,A -85,B 0,C 180,E1 -4178.948,E2 -4178.948} C_VEL
LIN {X 0,Y 532.029,Z 526.611,A -85,B 0,C 180,E1 -4179.407,E2 -4179.407} C_VEL
LIN {X 0,Y 531.772,Z 539.112,A -85,B 0,C 180,E1 -4180.046,E2 -4180.046} C_VEL
LIN {X 0,Y 531.543,Z 549.892,A -85,B 0,C 180,E1 -4180.756,E2 -4180.756} C_VEL
LIN {X 0,Y 531.202,Z 560.93,A -85,B 0,C 180,E1 -4181.669,E2 -4181.669} C_VEL
LIN {X 0,Y 530.997,Z 570.514,A -85,B 0,C 180,E1 -4182.657,E2 -4182.657} C_VEL
LIN {X 0,Y 530.805,Z 578.877,A -85,B 0,C 180,E1 -4183.717,E2 -4183.717} C_VEL
LIN {X 0,Y 530.633,Z 586.909,A -85,B 0,C 180,E1 -4184.995,E2 -4184.995} C_VEL
LIN {X 0,Y 530.572,Z 592.283,A -85,B 0,C 180,E1 -4186.066,E2 -4186.066} C_VEL
LIN {X 0,Y 530.52,Z 596.571,A -85,B 0,C 180,E1 -4187.132,E2 -4187.132} C_VEL
LIN {X 0,Y 530.462,Z 600.755,A -85,B 0,C 180,E1 -4188.513,E2 -4188.513} C_VEL
LIN {X 0,Y 530.364,Z 602.845,A -85,B 0,C 180,E1 -4189.509,E2 -4189.509} C_VEL
LIN {X 0,Y 530.362,Z 604.225,A -85,B 0,C 180,E1 -4190.5,E2 -4190.5} C_VEL
LIN {X 0,Y 530.343,Z 604.951,A -85,B 0,C 180,E1 -4191.476,E2 -4191.476} C_VEL
LIN {X 0,Y 530.342,Z 604.93,A -85,B 0,C 180,E1 -4192.666,E2 -4192.666} C_VEL
LIN {X 0,Y 530.344,Z 603.828,A -85,B 0,C 180,E1 -4193.936,E2 -4193.936} C_VEL
LIN {X 0,Y 530.412,Z 601.463,A -85,B 0,C 180,E1 -4195.266,E2 -4195.266} C_VEL
LIN {X 0,Y 530.48,Z 597.865,A -85,B 0,C 180,E1 -4196.58,E2 -4196.58} C_VEL
LIN {X 0,Y 530.573,Z 592.369,A -85,B 0,C 180,E1 -4198.004,E2 -4198.004} C_VEL
LIN {X 0,Y 530.67,Z 586.392,A -85,B 0,C 180,E1 -4199.185,E2 -4199.185} C_VEL
LIN {X 0,Y 530.853,Z 578.304,A -85,B 0,C 180,E1 -4200.451,E2 -4200.451} C_VEL
LIN {X 0,Y 531.048,Z 569.479,A -85,B 0,C 180,E1 -4201.547,E2 -4201.547} C_VEL
LIN {X 0,Y 531.27,Z 560.117,A -85,B 0,C 180,E1 -4202.494,E2 -4202.494} C_VEL
LIN {X 0,Y 531.558,Z 549.19,A -85,B 0,C 180,E1 -4203.383,E2 -4203.383} C_VEL
LIN {X 0,Y 531.811,Z 537.364,A -85,B 0,C 180,E1 -4204.144,E2 -4204.144} C_VEL
LIN {X 0,Y 532.05,Z 525.435,A -85,B 0,C 180,E1 -4204.733,E2 -4204.733} C_VEL
LIN {X 0,Y 532.271,Z 512.234,A -85,B 0,C 180,E1 -4205.204,E2 -4205.204} C_VEL
LIN {X 0,Y 532.424,Z 499.672,A -85,B 0,C 180,E1 -4205.498,E2 -4205.498} C_VEL
LIN {X 0,Y 532.747,Z 403.295,A -85,B 0,C 180,E1 -4206.814,E2 -4206.814} C_VEL
LIN {X 0,Y 531.196,Z 394.559,A -85,B 0,C 180,E1 -4207,E2 -4207} C_VEL
LIN {X 0,Y 531.565,Z 378.169,A -85,B 0,C 180,E1 -4210.095,E2 -4210.095} C_VEL
LIN {X 0,Y 531.571,Z 368.548,A -85,B 0,C 180,E1 -4211.938,E2 -4211.938} C_VEL
LIN {X 0,Y 531.064,Z 365.338,A -85,B 0,C 180,E1 -4212.617,E2 -4212.617} C_VEL
